KUKA KRL program: MyProgram_035().src

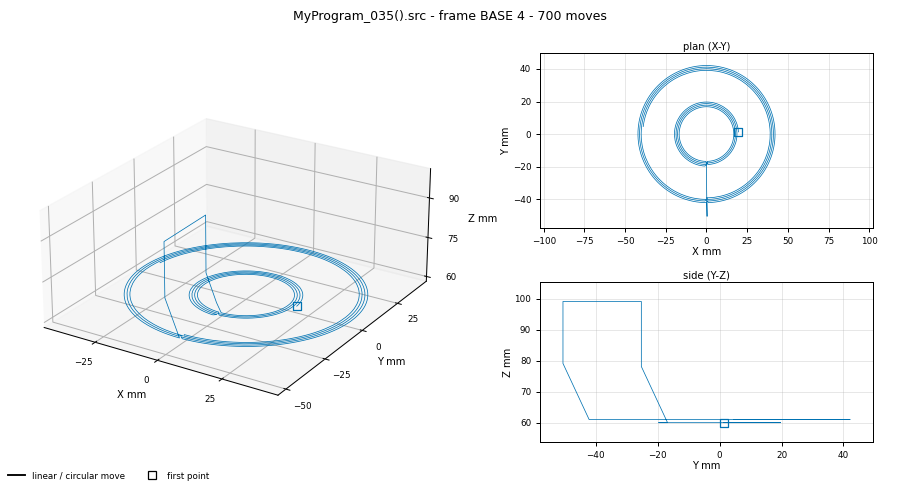
[picture p0: tool path of MyProgram_035().src in frame BASE 4, 700 of 700 moves have a stored position in this frame; points joined in program order, loops and branches not executed]
&ACCESS RVP
&REL 1
&PARAM TEMPLATE = C:\KRC\Roboter\Template\vorgabe
&PARAM EDITMASK = *
DEF MyProgram_035()
; ---- Setting reference (Base) ----
$BASE = BASE_DATA[4]

; --------------------------
; ---- Setting tool (TCP) ----
$TOOL = TOOL_DATA[3]
; --------------------------

$VEL.CP = VEL_APROX_PRINT
Startdeposition()
$VEL.CP = VEL_PRINT
LIN {X 19.6376,Y 1.3472,Z 60,A -3.0599,B 24.8058,C -3.2131,E1 25.1593,E2 -634.5538} C_DIS
LIN {X 19.5136,Y 2.5822,Z 60,A 0.9815,B 24.804,C -3.2283,E1 25.158,E2 -638.6073} C_DIS
LIN {X 19.2505,Y 4.1066,Z 60,A 5.5347,B 24.8023,C -3.2424,E1 25.1555,E2 -643.1673} C_DIS
LIN {X 18.8579,Y 5.6408,Z 60,A 9.7451,B 24.8011,C -3.2522,E1 25.1524,E2 -647.3767} C_DIS
LIN {X 18.3804,Y 7.044,Z 60,A 15.1354,B 24.7983,C -3.2746,E1 25.1472,E2 -652.7902} C_DIS
LIN {X 17.2808,Y 9.4251,Z 60,A 22.0117,B 24.7966,C -3.2881,E1 25.1387,E2 -659.6618} C_DIS
LIN {X 16.4135,Y 10.8654,Z 60,A 26.3437,B 24.7957,C -3.2954,E1 25.1323,E2 -663.9891} C_DIS
LIN {X 15.7405,Y 11.8191,Z 60,A 29.8972,B 24.7945,C -3.305,E1 25.1265,E2 -667.5481} C_DIS
LIN {X 14.7973,Y 12.9806,Z 60,A 34.6576,B 24.7928,C -3.3183,E1 25.1179,E2 -672.3185} C_DIS
LIN {X 13.3773,Y 14.4397,Z 60,A 40.2444,B 24.7917,C -3.3275,E1 25.1068,E2 -677.9036} C_DIS
LIN {X 12.4967,Y 15.2079,Z 60,A 44.9046,B 24.7896,C -3.3443,E1 25.0967,E2 -682.5859} C_DIS
LIN {X 10.1616,Y 16.8582,Z 60,A 52.5619,B 24.7886,C -3.3517,E1 25.0788,E2 -690.2355} C_DIS
LIN {X 8.1073,Y 17.9362,Z 60,A 58.7713,B 24.7881,C -3.3556,E1 25.0633,E2 -696.4376} C_DIS
LIN {X 6.6276,Y 18.5344,Z 60,A 63.8081,B 24.7872,C -3.3628,E1 25.0502,E2 -701.4806} C_DIS
LIN {X 4.5052,Y 19.1613,Z 60,A 69.8964,B 24.787,C -3.3643,E1 25.0338,E2 -707.5628} C_DIS
LIN {X 3.2717,Y 19.4101,Z 60,A 73.6602,B 24.7868,C -3.3663,E1 25.0234,E2 -711.3272} C_DIS
LIN {X 1.6592,Y 19.6136,Z 60,A 78.087,B 24.7869,C -3.365,E1 25.0112,E2 -715.7478} C_DIS
LIN {X 0.0594,Y 19.6839,Z 60,A 83.0982,B 24.7867,C -3.3666,E1 24.9972,E2 -720.7621} C_DIS
LIN {X -1.6521,Y 19.6141,Z 60,A 87.634,B 24.7873,C -3.362,E1 24.9846,E2 -725.2883} C_DIS
LIN {X -2.7882,Y 19.4854,Z 60,A 91.6136,B 24.7871,C -3.3639,E1 24.9735,E2 -729.2752} C_DIS
LIN {X -4.6137,Y 19.1352,Z 60,A 96.3255,B 24.7882,C -3.3554,E1 24.9607,E2 -733.9727} C_DIS
LIN {X -5.6169,Y 18.8652,Z 60,A 99.3541,B 24.7886,C -3.3523,E1 24.9526,E2 -736.9987} C_DIS
LIN {X -6.5937,Y 18.5466,Z 60,A 102.691,B 24.7888,C -3.3506,E1 24.9437,E2 -740.3378} C_DIS
LIN {X -7.8497,Y 18.0506,Z 60,A 106.9874,B 24.7892,C -3.347,E1 24.9327,E2 -744.6356} C_DIS
LIN {X -9.2709,Y 17.3642,Z 60,A 111.6347,B 24.7901,C -3.3399,E1 24.9212,E2 -749.2786} C_DIS
LIN {X -11.1212,Y 16.2413,Z 60,A 118.0633,B 24.7915,C -3.3289,E1 24.9061,E2 -755.7015} C_DIS
LIN {X -12.8725,Y 14.8916,Z 60,A 124.2464,B 24.7934,C -3.3142,E1 24.8927,E2 -761.8727} C_DIS
LIN {X -14.1296,Y 13.7045,Z 60,A 129.3126,B 24.7948,C -3.3026,E1 24.8827,E2 -766.9325} C_DIS
LIN {X -15.2762,Y 12.4134,Z 60,A 134.329,B 24.7964,C -3.2901,E1 24.8736,E2 -771.9417} C_DIS
LIN {X -16.2565,Y 11.099,Z 60,A 139.6568,B 24.7977,C -3.2795,E1 24.865,E2 -777.2704} C_DIS
LIN {X -17.4357,Y 9.1344,Z 60,A 145.3666,B 24.8004,C -3.2573,E1 24.8572,E2 -782.9568} C_DIS
LIN {X -17.9124,Y 8.1607,Z 60,A 149.1514,B 24.8013,C -3.2504,E1 24.8527,E2 -786.7456} C_DIS
LIN {X -18.4403,Y 6.8842,Z 60,A 152.9543,B 24.8028,C -3.2377,E1 24.8489,E2 -790.5395} C_DIS
LIN {X -18.9649,Y 5.2698,Z 60,A 158.2599,B 24.8045,C -3.224,E1 24.8446,E2 -795.8427} C_DIS
LIN {X -19.4015,Y 3.3237,Z 60,A 162.9983,B 24.8071,C -3.2024,E1 24.8419,E2 -800.5574} C_DIS
LIN {X -19.5797,Y 2.0215,Z 60,A 167.8103,B 24.8082,C -3.1938,E1 24.8403,E2 -805.3776} C_DIS
LIN {X -19.6813,Y 0.325,Z 60,A 172.3497,B 24.8102,C -3.177,E1 24.8398,E2 -809.904} C_DIS
LIN {X -19.638,Y -1.3384,Z 60,A 178.2471,B 24.8115,C -3.1657,E1 24.8406,E2 -815.8097} C_DIS
LIN {X -19.2559,Y -4.0801,Z 60,A -173.6054,B 24.8144,C -3.1416,E1 24.8445,E2 -823.9478} C_DIS
LIN {X -18.7721,Y -5.9197,Z 60,A -168.9163,B 24.8167,C -3.1223,E1 24.8481,E2 -828.6178} C_DIS
LIN {X -18.3574,Y -7.1031,Z 60,A -165.3994,B 24.818,C -3.1114,E1 24.8515,E2 -832.1285} C_DIS
LIN {X -17.8438,Y -8.3091,Z 60,A -161.3071,B 24.8191,C -3.102,E1 24.8561,E2 -836.2206} C_DIS
LIN {X -17.2608,Y -9.4618,Z 60,A -157.8679,B 24.8204,C -3.0907,E1 24.8606,E2 -839.6513} C_DIS
LIN {X -16.491,Y -10.7477,Z 60,A -152.7383,B 24.8213,C -3.0828,E1 24.8682,E2 -844.788} C_DIS
LIN {X -15.6196,Y -11.978,Z 60,A -148.4735,B 24.8226,C -3.0719,E1 24.8753,E2 -849.0473} C_DIS
LIN {X -14.4508,Y -13.3656,Z 60,A -143.6937,B 24.8242,C -3.0581,E1 24.8841,E2 -853.8156} C_DIS
LIN {X -13.2063,Y -14.5954,Z 60,A -138.0741,B 24.8251,C -3.0504,E1 24.8955,E2 -859.44} C_DIS
LIN {X -11.8732,Y -15.6997,Z 60,A -133.0339,B 24.8261,C -3.0416,E1 24.9065,E2 -864.4776} C_DIS
LIN {X -10.7284,Y -16.5033,Z 60,A -129.3592,B 24.8271,C -3.0333,E1 24.915,E2 -868.1447} C_DIS
LIN {X -9.4145,Y -17.2865,Z 60,A -124.345,B 24.8274,C -3.0302,E1 24.9272,E2 -873.1664} C_DIS
LIN {X -7.5215,Y -18.1901,Z 60,A -119.2037,B 24.8288,C -3.0183,E1 24.9402,E2 -878.2918} C_DIS
LIN {X -6.3703,Y -18.6242,Z 60,A -114.7625,B 24.8286,C -3.0202,E1 24.9519,E2 -882.7465} C_DIS
LIN {X -4.7968,Y -19.0901,Z 60,A -109.6924,B 24.8286,C -3.0191,E1 24.9656,E2 -887.8218} C_DIS
LIN {X -2.3633,Y -19.5413,Z 60,A -103.3398,B 24.8295,C -3.0117,E1 24.983,E2 -894.1625} C_DIS
LIN {X -0.9908,Y -19.6586,Z 60,A -98.6362,B 24.829,C -3.0163,E1 24.9962,E2 -898.879} C_DIS
LIN {X -0.9908,Y -19.6586,Z 60,A -98.6362,B 24.829,C -3.0163,E1 24.9962,E2 -898.879} C_DIS
Enddeposition()
LIN {X 0.0023,Y -18.7203,Z 60,A -97.1672,B 24.8281,C -3.024,E1 25.0003,E2 -900.3662} C_DIS
Startdeposition()
$VEL.CP = VEL_PRINT
LIN {X -1.3074,Y -18.6798,Z 60,A -102.4252,B 24.829,C -3.0158,E1 24.9856,E2 -895.0876} C_DIS
LIN {X -2.9728,Y -18.4887,Z 60,A -107.3213,B 24.8288,C -3.0182,E1 24.9721,E2 -890.1933} C_DIS
LIN {X -4.4742,Y -18.1833,Z 60,A -112.0588,B 24.8286,C -3.02,E1 24.9591,E2 -885.4543} C_DIS
LIN {X -5.7912,Y -17.8071,Z 60,A -116.0247,B 24.8281,C -3.0241,E1 24.9486,E2 -881.4913} C_DIS
LIN {X -7.2175,Y -17.2787,Z 60,A -120.3356,B 24.8274,C -3.0301,E1 24.9373,E2 -877.1856} C_DIS
LIN {X -8.0909,Y -16.8875,Z 60,A -124.1301,B 24.8275,C -3.0291,E1 24.9277,E2 -873.3792} C_DIS
LIN {X -9.7048,Y -16.0147,Z 60,A -129.7588,B 24.8267,C -3.0366,E1 24.9141,E2 -867.7519} C_DIS
LIN {X -11.1863,Y -15.0175,Z 60,A -135.1337,B 24.8256,C -3.0458,E1 24.9018,E2 -862.3804} C_DIS
LIN {X -12.5346,Y -13.912,Z 60,A -140.552,B 24.8245,C -3.0554,E1 24.8903,E2 -856.9639} C_DIS
LIN {X -13.7315,Y -12.7322,Z 60,A -145.7596,B 24.8233,C -3.0658,E1 24.8802,E2 -851.7589} C_DIS
LIN {X -14.7656,Y -11.5172,Z 60,A -151.4599,B 24.8224,C -3.074,E1 24.8703,E2 -846.0516} C_DIS
LIN {X -16.3018,Y -9.215,Z 60,A -159.7556,B 24.8198,C -3.096,E1 24.8581,E2 -837.7662} C_DIS
LIN {X -17.2394,Y -7.3112,Z 60,A -165.587,B 24.8175,C -3.1159,E1 24.8513,E2 -831.9507} C_DIS
LIN {X -17.7997,Y -5.8135,Z 60,A -170.3075,B 24.8157,C -3.1305,E1 24.8469,E2 -827.2382} C_DIS
LIN {X -18.199,Y -4.4089,Z 60,A -175.0055,B 24.8143,C -3.143,E1 24.8436,E2 -822.5429} C_DIS
LIN {X -18.4596,Y -3.1467,Z 60,A -178.7025,B 24.8128,C -3.1556,E1 24.8417,E2 -818.8542} C_DIS
LIN {X -18.6406,Y -1.7791,Z 60,A 176.7274,B 24.8113,C -3.1675,E1 24.8402,E2 -814.2853} C_DIS
LIN {X -18.7241,Y 0.0458,Z 60,A 171.3284,B 24.8092,C -3.1854,E1 24.8398,E2 -808.8967} C_DIS
LIN {X -18.6556,Y 1.6172,Z 60,A 166.2101,B 24.8075,C -3.1995,E1 24.8407,E2 -803.7814} C_DIS
LIN {X -18.4421,Y 3.248,Z 60,A 161.0802,B 24.8056,C -3.2149,E1 24.8429,E2 -798.6578} C_DIS
LIN {X -18.0417,Y 5.0134,Z 60,A 155.5596,B 24.8035,C -3.2319,E1 24.8466,E2 -793.1458} C_DIS
LIN {X -17.4548,Y 6.7805,Z 60,A 150.3263,B 24.8013,C -3.2504,E1 24.8514,E2 -787.927} C_DIS
LIN {X -17.0487,Y 7.7456,Z 60,A 146.7149,B 24.8003,C -3.2585,E1 24.8555,E2 -784.3152} C_DIS
LIN {X -16.289,Y 9.2368,Z 60,A 140.7953,B 24.7988,C -3.2705,E1 24.8634,E2 -778.3931} C_DIS
LIN {X -15.1642,Y 10.9866,Z 60,A 135.0172,B 24.7964,C -3.2895,E1 24.8724,E2 -772.6318} C_DIS
LIN {X -14.128,Y 12.2906,Z 60,A 129.8754,B 24.7949,C -3.3021,E1 24.8816,E2 -767.4966} C_DIS
LIN {X -12.9816,Y 13.4956,Z 60,A 124.7751,B 24.7934,C -3.314,E1 24.8916,E2 -762.403} C_DIS
LIN {X -11.9092,Y 14.451,Z 60,A 120.0573,B 24.7923,C -3.3223,E1 24.9017,E2 -757.6868} C_DIS
LIN {X -10.4305,Y 15.552,Z 60,A 114.9908,B 24.7907,C -3.3356,E1 24.9131,E2 -752.6347} C_DIS
LIN {X -9.0786,Y 16.3779,Z 60,A 109.8141,B 24.7898,C -3.3426,E1 24.9256,E2 -747.4592} C_DIS
LIN {X -7.5346,Y 17.1427,Z 60,A 104.2599,B 24.7889,C -3.3492,E1 24.9397,E2 -741.907} C_DIS
LIN {X -5.6024,Y 17.8678,Z 60,A 97.8473,B 24.788,C -3.3563,E1 24.9566,E2 -735.499} C_DIS
LIN {X -3.4857,Y 18.3984,Z 60,A 91.502,B 24.7871,C -3.3638,E1 24.9738,E2 -729.1635} C_DIS
LIN {X -1.8213,Y 18.6369,Z 60,A 86.2377,B 24.7868,C -3.3661,E1 24.9884,E2 -723.901} C_DIS
LIN {X -0.1445,Y 18.7253,Z 60,A 81.1999,B 24.7865,C -3.3681,E1 25.0025,E2 -718.8673} C_DIS
LIN {X 1.3917,Y 18.6736,Z 60,A 76.1915,B 24.7868,C -3.3664,E1 25.0164,E2 -713.8567} C_DIS
LIN {X 3.3103,Y 18.4309,Z 60,A 70.337,B 24.7869,C -3.3651,E1 25.0326,E2 -708.0047} C_DIS
LIN {X 5.2188,Y 17.9836,Z 60,A 64.4223,B 24.7873,C -3.3621,E1 25.0485,E2 -702.0919} C_DIS
LIN {X 6.6991,Y 17.4858,Z 60,A 60.4332,B 24.7871,C -3.3634,E1 25.059,E2 -698.1141} C_DIS
LIN {X 7.7404,Y 17.051,Z 60,A 56.5752,B 24.788,C -3.3568,E1 25.0689,E2 -694.2498} C_DIS
LIN {X 8.9291,Y 16.4598,Z 60,A 52.631,B 24.7885,C -3.3526,E1 25.0787,E2 -690.3065} C_DIS
LIN {X 10.4844,Y 15.515,Z 60,A 45.6574,B 24.7909,C -3.3336,E1 25.0951,E2 -683.3106} C_DIS
LIN {X 12.3955,Y 14.0359,Z 60,A 39.895,B 24.791,C -3.3329,E1 25.1075,E2 -677.5682} C_DIS
LIN {X 13.3706,Y 13.1097,Z 60,A 35.602,B 24.7922,C -3.3231,E1 25.116,E2 -673.27} C_DIS
LIN {X 14.248,Y 12.1511,Z 60,A 31.5215,B 24.7934,C -3.3135,E1 25.1236,E2 -669.185} C_DIS
LIN {X 15.218,Y 10.912,Z 60,A 26.5171,B 24.7951,C -3.3005,E1 25.132,E2 -664.1737} C_DIS
LIN {X 16.1415,Y 9.4927,Z 60,A 21.3329,B 24.7967,C -3.2873,E1 25.1396,E2 -658.9845} C_DIS
LIN {X 16.9883,Y 7.8764,Z 60,A 15.6192,B 24.7987,C -3.2711,E1 25.1467,E2 -653.2629} C_DIS
LIN {X 17.5234,Y 6.6008,Z 60,A 11.2667,B 24.8003,C -3.2581,E1 25.1511,E2 -648.9037} C_DIS
LIN {X 18.1197,Y 4.7245,Z 60,A 5.6681,B 24.802,C -3.2442,E1 25.1555,E2 -643.3042} C_DIS
LIN {X 18.4918,Y 2.9509,Z 60,A -0.4867,B 24.8048,C -3.222,E1 25.1585,E2 -637.1327} C_DIS
LIN {X 18.704,Y 0.8956,Z 60,A -6.4334,B 24.8067,C -3.2058,E1 25.1597,E2 -631.1831} C_DIS
LIN {X 18.7034,Y -0.9078,Z 60,A -11.3548,B 24.8081,C -3.1941,E1 25.1594,E2 -626.2631} C_DIS
LIN {X 18.5918,Y -2.2333,Z 60,A -15.3986,B 24.8096,C -3.1816,E1 25.1583,E2 -622.2138} C_DIS
LIN {X 18.3067,Y -3.9382,Z 60,A -20.8999,B 24.8118,C -3.1633,E1 25.1555,E2 -616.7012} C_DIS
LIN {X 17.8954,Y -5.5135,Z 60,A -25.9073,B 24.8137,C -3.1478,E1 25.1516,E2 -611.6858} C_DIS
LIN {X 17.4696,Y -6.7422,Z 60,A -29.5087,B 24.8147,C -3.1393,E1 25.1481,E2 -608.0844} C_DIS
LIN {X 17.0745,Y -7.6882,Z 60,A -32.8176,B 24.816,C -3.1286,E1 25.1444,E2 -604.768} C_DIS
LIN {X 16.3664,Y -9.0987,Z 60,A -37.4347,B 24.8174,C -3.1166,E1 25.1384,E2 -600.147} C_DIS
LIN {X 15.6588,Y -10.2663,Z 60,A -40.6077,B 24.8177,C -3.114,E1 25.1338,E2 -596.9839} C_DIS
LIN {X 15.164,Y -10.9869,Z 60,A -44.1903,B 24.8195,C -3.0988,E1 25.128,E2 -593.3828} C_DIS
LIN {X 14.3596,Y -12.0187,Z 60,A -48.9247,B 24.8214,C -3.0823,E1 25.1196,E2 -588.6312} C_DIS
LIN {X 13.0169,Y -13.4616,Z 60,A -54.4704,B 24.8226,C -3.072,E1 25.1088,E2 -583.0849} C_DIS
LIN {X 11.6539,Y -14.6571,Z 60,A -59.971,B 24.8239,C -3.0604,E1 25.097,E2 -577.5777} C_DIS
LIN {X 10.4375,Y -15.5473,Z 60,A -64.481,B 24.8249,C -3.0521,E1 25.0867,E2 -573.0636} C_DIS
LIN {X 9.1733,Y -16.3247,Z 60,A -69.5837,B 24.8263,C -3.0397,E1 25.0744,E2 -567.947} C_DIS
LIN {X 7.4057,Y -17.1987,Z 60,A -75.1897,B 24.827,C -3.0338,E1 25.0602,E2 -562.3413} C_DIS
LIN {X 5.9027,Y -17.7706,Z 60,A -79.0907,B 24.8269,C -3.035,E1 25.05,E2 -558.4513} C_DIS
LIN {X 4.7432,Y -18.1147,Z 60,A -84.1337,B 24.8284,C -3.0215,E1 25.0364,E2 -553.3845} C_DIS
LIN {X 2.5879,Y -18.546,Z 60,A -90.5837,B 24.8288,C -3.0183,E1 25.0186,E2 -546.9337} C_DIS
LIN {X 0.9263,Y -18.7024,Z 60,A -95.0252,B 24.8285,C -3.0203,E1 25.0063,E2 -542.4991} C_DIS
LIN {X 0.9263,Y -18.7024,Z 60,A -95.0252,B 24.8285,C -3.0203,E1 25.0063,E2 -542.4991} C_DIS
Enddeposition()
LIN {X 0.0155,Y -17.7649,Z 60,A -97.9923,B 24.8268,C -3.0353,E1 24.9981,E2 -539.5681} C_DIS
Startdeposition()
$VEL.CP = VEL_PRINT
LIN {X 0.9859,Y -17.7401,Z 60,A -92.6978,B 24.8252,C -3.0497,E1 25.013,E2 -544.8957} C_DIS
LIN {X 2.8059,Y -17.5446,Z 60,A -86.903,B 24.8248,C -3.0527,E1 25.029,E2 -550.6929} C_DIS
LIN {X 4.419,Y -17.2087,Z 60,A -82.0027,B 24.8246,C -3.0547,E1 25.0423,E2 -555.5912} C_DIS
LIN {X 5.782,Y -16.8003,Z 60,A -76.9277,B 24.8236,C -3.0635,E1 25.0559,E2 -560.6777} C_DIS
LIN {X 7.3313,Y -16.1845,Z 60,A -71.5706,B 24.8227,C -3.0711,E1 25.0696,E2 -566.0401} C_DIS
LIN {X 8.8093,Y -15.4301,Z 60,A -66.2939,B 24.8217,C -3.0795,E1 25.0826,E2 -571.3216} C_DIS
LIN {X 10.1378,Y -14.5916,Z 60,A -61.2643,B 24.8206,C -3.0889,E1 25.0943,E2 -576.3567} C_DIS
LIN {X 11.4347,Y -13.5993,Z 60,A -55.9441,B 24.8193,C -3.1005,E1 25.1059,E2 -581.6845} C_DIS
LIN {X 12.6468,Y -12.4798,Z 60,A -50.6998,B 24.8179,C -3.1122,E1 25.1164,E2 -586.9349} C_DIS
LIN {X 13.7519,Y -11.2508,Z 60,A -45.3857,B 24.8163,C -3.1254,E1 25.1261,E2 -592.2562} C_DIS
LIN {X 14.48,Y -10.2967,Z 60,A -41.3387,B 24.8149,C -3.1372,E1 25.1328,E2 -596.3116} C_DIS
LIN {X 15.3947,Y -8.871,Z 60,A -36.4867,B 24.8138,C -3.147,E1 25.1398,E2 -601.1622} C_DIS
LIN {X 15.9584,Y -7.8103,Z 60,A -32.2515,B 24.8121,C -3.1614,E1 25.1452,E2 -605.4089} C_DIS
LIN {X 16.6204,Y -6.2801,Z 60,A -26.9211,B 24.8102,C -3.1769,E1 25.1508,E2 -610.7467} C_DIS
LIN {X 17.1291,Y -4.7193,Z 60,A -21.6748,B 24.8083,C -3.1926,E1 25.155,E2 -616.0002} C_DIS
LIN {X 17.4958,Y -3.0967,Z 60,A -16.5828,B 24.8066,C -3.2067,E1 25.1578,E2 -621.096} C_DIS
LIN {X 17.6916,Y -1.6394,Z 60,A -11.8559,B 24.8048,C -3.2214,E1 25.1593,E2 -625.8297} C_DIS
LIN {X 17.7588,Y -0.5555,Z 60,A -7.9269,B 24.803,C -3.2362,E1 25.1598,E2 -629.7704} C_DIS
LIN {X 17.7238,Y 1.2423,Z 60,A -2.3861,B 24.8011,C -3.2518,E1 25.1591,E2 -635.3153} C_DIS
LIN {X 17.5367,Y 2.8563,Z 60,A 2.8447,B 24.7991,C -3.2677,E1 25.1571,E2 -640.553} C_DIS
LIN {X 17.0145,Y 5.1185,Z 60,A 11.2683,B 24.7954,C -3.2982,E1 25.151,E2 -649.0004} C_DIS
LIN {X 16.2621,Y 7.1575,Z 60,A 17.5108,B 24.7937,C -3.3111,E1 25.1444,E2 -655.239} C_DIS
LIN {X 15.4456,Y 8.7823,Z 60,A 23.048,B 24.7922,C -3.3238,E1 25.1371,E2 -660.7772} C_DIS
LIN {X 14.5893,Y 10.1411,Z 60,A 28.1705,B 24.7906,C -3.3361,E1 25.1292,E2 -665.9036} C_DIS
LIN {X 13.5375,Y 11.5077,Z 60,A 33.9985,B 24.7887,C -3.3511,E1 25.1189,E2 -671.7401} C_DIS
LIN {X 12.2964,Y 12.8253,Z 60,A 39.5523,B 24.7875,C -3.3609,E1 25.108,E2 -677.2934} C_DIS
LIN {X 11.0852,Y 13.8857,Z 60,A 44.6875,B 24.7863,C -3.37,E1 25.097,E2 -682.4306} C_DIS
LIN {X 9.7729,Y 14.8385,Z 60,A 49.6403,B 24.7855,C -3.3764,E1 25.0857,E2 -687.3815} C_DIS
LIN {X 8.5658,Y 15.5668,Z 60,A 54.8686,B 24.7841,C -3.3875,E1 25.073,E2 -692.6209} C_DIS
LIN {X 6.8255,Y 16.4041,Z 60,A 60.4967,B 24.7837,C -3.3902,E1 25.0587,E2 -698.2412} C_DIS
LIN {X 5.1776,Y 16.9963,Z 60,A 66.6407,B 24.7827,C -3.398,E1 25.0424,E2 -704.392} C_DIS
LIN {X 3.6988,Y 17.3781,Z 60,A 70.4944,B 24.7833,C -3.3937,E1 25.032,E2 -708.2302} C_DIS
LIN {X 2.1269,Y 17.6396,Z 60,A 76.3306,B 24.7825,C -3.3994,E1 25.0158,E2 -714.0744} C_DIS
LIN {X 0.5104,Y 17.7602,Z 60,A 81.5201,B 24.7825,C -3.399,E1 25.0014,E2 -719.2612} C_DIS
LIN {X -1.0448,Y 17.7365,Z 60,A 86.6495,B 24.7827,C -3.3981,E1 24.9871,E2 -724.3894} C_DIS
LIN {X -2.7119,Y 17.5595,Z 60,A 92.0361,B 24.7831,C -3.3948,E1 24.9722,E2 -729.772} C_DIS
LIN {X -4.288,Y 17.2422,Z 60,A 97.2456,B 24.7837,C -3.3904,E1 24.958,E2 -734.9777} C_DIS
LIN {X -5.3974,Y 16.9275,Z 60,A 101.2596,B 24.784,C -3.3877,E1 24.9473,E2 -738.9922} C_DIS
LIN {X -7.2707,Y 16.2117,Z 60,A 107.9497,B 24.785,C -3.3798,E1 24.9301,E2 -745.6788} C_DIS
LIN {X -8.9768,Y 15.3334,Z 60,A 112.926,B 24.787,C -3.3645,E1 24.9179,E2 -750.6325} C_DIS
LIN {X -9.8381,Y 14.7955,Z 60,A 116.3784,B 24.7877,C -3.3592,E1 24.9098,E2 -754.0832} C_DIS
LIN {X -10.8797,Y 14.0472,Z 60,A 121.1427,B 24.7884,C -3.3532,E1 24.8991,E2 -758.8504} C_DIS
LIN {X -12.1249,Y 12.9875,Z 60,A 126.3848,B 24.7899,C -3.3415,E1 24.8882,E2 -764.0852} C_DIS
LIN {X -13.2496,Y 11.838,Z 60,A 131.6257,B 24.7915,C -3.3292,E1 24.8782,E2 -769.3195} C_DIS
LIN {X -14.2665,Y 10.5908,Z 60,A 136.8701,B 24.7931,C -3.316,E1 24.8693,E2 -774.5573} C_DIS
LIN {X -15.1697,Y 9.2502,Z 60,A 141.9423,B 24.795,C -3.3014,E1 24.8616,E2 -779.6201} C_DIS
LIN {X -15.8004,Y 8.1265,Z 60,A 145.8324,B 24.7965,C -3.2888,E1 24.8565,E2 -783.5006} C_DIS
LIN {X -16.3391,Y 6.9794,Z 60,A 150.1115,B 24.7979,C -3.2775,E1 24.8516,E2 -787.776} C_DIS
LIN {X -16.8888,Y 5.518,Z 60,A 155.9725,B 24.7995,C -3.2648,E1 24.8462,E2 -793.6399} C_DIS
LIN {X -17.3922,Y 3.6333,Z 60,A 161.8048,B 24.802,C -3.2441,E1 24.8425,E2 -799.4568} C_DIS
LIN {X -17.6508,Y 2.0329,Z 60,A 167.1192,B 24.804,C -3.2281,E1 24.8404,E2 -804.7647} C_DIS
LIN {X -17.764,Y 0.3659,Z 60,A 172.7123,B 24.806,C -3.2119,E1 24.8398,E2 -810.3525} C_DIS
LIN {X -17.7434,Y -0.9139,Z 60,A 176.7278,B 24.8076,C -3.1989,E1 24.8402,E2 -814.3608} C_DIS
LIN {X -17.5864,Y -2.5306,Z 60,A -177.5893,B 24.8093,C -3.1841,E1 24.8422,E2 -820.0423} C_DIS
LIN {X -17.0785,Y -4.8999,Z 60,A -170.2362,B 24.8123,C -3.1595,E1 24.847,E2 -827.3795} C_DIS
LIN {X -16.569,Y -6.4147,Z 60,A -165.0333,B 24.814,C -3.145,E1 24.852,E2 -832.577} C_DIS
LIN {X -16.046,Y -7.6299,Z 60,A -161.0987,B 24.8155,C -3.1322,E1 24.8565,E2 -836.5026} C_DIS
LIN {X -15.4602,Y -8.7566,Z 60,A -156.7355,B 24.8167,C -3.1223,E1 24.8623,E2 -840.8652} C_DIS
LIN {X -14.767,Y -9.88,Z 60,A -151.9945,B 24.8178,C -3.1134,E1 24.8695,E2 -845.6087} C_DIS
LIN {X -13.685,Y -11.3319,Z 60,A -146.3624,B 24.8194,C -3.0992,E1 24.8792,E2 -851.2332} C_DIS
LIN {X -12.5761,Y -12.5515,Z 60,A -141.0401,B 24.8207,C -3.088,E1 24.8895,E2 -856.552} C_DIS
LIN {X -11.35,Y -13.67,Z 60,A -135.6464,B 24.8219,C -3.0782,E1 24.9008,E2 -861.9433} C_DIS
LIN {X -10.2593,Y -14.5066,Z 60,A -131.2588,B 24.8227,C -3.0706,E1 24.9107,E2 -866.3283} C_DIS
LIN {X -8.9005,Y -15.3776,Z 60,A -125.9838,B 24.8236,C -3.0635,E1 24.9233,E2 -871.6026} C_DIS
LIN {X -7.3207,Y -16.1892,Z 60,A -120.3803,B 24.8244,C -3.0563,E1 24.9374,E2 -877.2034} C_DIS
LIN {X -6.0534,Y -16.7038,Z 60,A -116.2283,B 24.825,C -3.051,E1 24.9482,E2 -881.3515} C_DIS
LIN {X -4.626,Y -17.1546,Z 60,A -111.0042,B 24.8251,C -3.0499,E1 24.9622,E2 -886.5816} C_DIS
LIN {X -3.0319,Y -17.5074,Z 60,A -105.7637,B 24.8254,C -3.0477,E1 24.9765,E2 -891.8228} C_DIS
LIN {X -1.4921,Y -17.7046,Z 60,A -100.694,B 24.8254,C -3.0477,E1 24.9906,E2 -896.8952} C_DIS
LIN {X 0.0155,Y -17.7649,Z 60,A -97.9922,B 24.8268,C -3.0353,E1 24.9981,E2 -899.5681} C_DIS
Enddeposition()
LIN {X 0.0155,Y -17.7649,Z 60,A -97.9922,B 24.8268,C -3.0353,E1 24.9981,E2 -899.5681} C_DIS
Startdeposition()
$VEL.CP = VEL_PRINT
LIN {X -0.4182,Y -16.8044,Z 60,A -100.0886,B 24.8253,C -3.0484,E1 24.9923,E2 -897.5028} C_DIS
LIN {X -1.9453,Y -16.6964,Z 60,A -105.0785,B 24.8251,C -3.05,E1 24.9785,E2 -892.514} C_DIS
LIN {X -3.3845,Y -16.4651,Z 60,A -110.07,B 24.825,C -3.0515,E1 24.9647,E2 -887.521} C_DIS
LIN {X -4.8682,Y -16.089,Z 60,A -115.4755,B 24.8247,C -3.0539,E1 24.9502,E2 -882.1125} C_DIS
LIN {X -6.509,Y -15.497,Z 60,A -119.9286,B 24.8233,C -3.0659,E1 24.9386,E2 -877.6791} C_DIS
LIN {X -7.8899,Y -14.8426,Z 60,A -125.1752,B 24.8226,C -3.0716,E1 24.9254,E2 -872.4327} C_DIS
LIN {X -9.2418,Y -14.0409,Z 60,A -130.6854,B 24.8218,C -3.0784,E1 24.9121,E2 -866.9222} C_DIS
LIN {X -10.5128,Y -13.1165,Z 60,A -136.1827,B 24.8209,C -3.0867,E1 24.8997,E2 -861.4255} C_DIS
LIN {X -11.2936,Y -12.4505,Z 60,A -140.4226,B 24.8204,C -3.0906,E1 24.8908,E2 -857.1782} C_DIS
LIN {X -12.2148,Y -11.548,Z 60,A -145.3533,B 24.8196,C -3.0979,E1 24.8811,E2 -852.2439} C_DIS
LIN {X -13.2504,Y -10.344,Z 60,A -150.6717,B 24.8181,C -3.1105,E1 24.8717,E2 -846.9309} C_DIS
LIN {X -13.8659,Y -9.5027,Z 60,A -153.9519,B 24.817,C -3.1199,E1 24.8664,E2 -843.6571} C_DIS
LIN {X -14.7157,Y -8.1246,Z 60,A -158.512,B 24.815,C -3.1367,E1 24.8599,E2 -839.1139} C_DIS
LIN {X -15.0377,Y -7.5116,Z 60,A -161.937,B 24.8146,C -3.1401,E1 24.8555,E2 -835.6786} C_DIS
LIN {X -15.6146,Y -6.2234,Z 60,A -167.1215,B 24.8131,C -3.1525,E1 24.8498,E2 -830.4951} C_DIS
LIN {X -16.144,Y -4.6824,Z 60,A -172.7406,B 24.8112,C -3.1684,E1 24.8451,E2 -824.882} C_DIS
LIN {X -16.5214,Y -3.0984,Z 60,A -178.1227,B 24.8092,C -3.1854,E1 24.842,E2 -819.5089} C_DIS
LIN {X -16.7334,Y -1.5956,Z 60,A 176.546,B 24.8073,C -3.2009,E1 24.8402,E2 -814.1829} C_DIS
LIN {X -16.8079,Y -0.1139,Z 60,A 171.6038,B 24.8054,C -3.2169,E1 24.8398,E2 -809.2491} C_DIS
LIN {X -16.7476,Y 1.4383,Z 60,A 166.1857,B 24.8034,C -3.2331,E1 24.8407,E2 -803.8373} C_DIS
LIN {X -16.5501,Y 2.9418,Z 60,A 162.0715,B 24.8011,C -3.2515,E1 24.8423,E2 -799.7428} C_DIS
LIN {X -16.1968,Y 4.4952,Z 60,A 156.6454,B 24.7991,C -3.2682,E1 24.8457,E2 -794.3248} C_DIS
LIN {X -15.9948,Y 5.1686,Z 60,A 153.1141,B 24.7985,C -3.2728,E1 24.8486,E2 -790.7842} C_DIS
LIN {X -15.4869,Y 6.5352,Z 60,A 148.1021,B 24.7967,C -3.2874,E1 24.8538,E2 -785.7792} C_DIS
LIN {X -14.7754,Y 8.0154,Z 60,A 143.6108,B 24.7944,C -3.3062,E1 24.8593,E2 -781.3089} C_DIS
LIN {X -13.9899,Y 9.319,Z 60,A 138.2998,B 24.7926,C -3.3202,E1 24.867,E2 -776.0042} C_DIS
LIN {X -13.4314,Y 10.1073,Z 60,A 133.758,B 24.7919,C -3.3255,E1 24.8745,E2 -771.4528} C_DIS
LIN {X -12.4167,Y 11.3305,Z 60,A 128.4235,B 24.7902,C -3.3391,E1 24.8842,E2 -766.1269} C_DIS
LIN {X -11.168,Y 12.5634,Z 60,A 123.5433,B 24.7881,C -3.3562,E1 24.894,E2 -761.2674} C_DIS
LIN {X -9.9444,Y 13.5524,Z 60,A 118.2043,B 24.7866,C -3.3675,E1 24.9056,E2 -755.9355} C_DIS
LIN {X -8.6339,Y 14.423,Z 60,A 112.715,B 24.7854,C -3.3771,E1 24.9183,E2 -750.4512} C_DIS
LIN {X -7.2839,Y 15.1493,Z 60,A 107.5379,B 24.7843,C -3.3859,E1 24.9311,E2 -745.2805} C_DIS
LIN {X -6.6823,Y 15.4237,Z 60,A 104.0355,B 24.7845,C -3.3842,E1 24.94,E2 -741.7656} C_DIS
LIN {X -5.2567,Y 15.966,Z 60,A 99.1574,B 24.7835,C -3.3919,E1 24.9528,E2 -736.8963} C_DIS
LIN {X -3.7006,Y 16.3971,Z 60,A 94.4476,B 24.7824,C -3.4008,E1 24.9655,E2 -732.2006} C_DIS
LIN {X -2.6638,Y 16.5974,Z 60,A 90.1413,B 24.7824,C -3.4002,E1 24.9773,E2 -727.8884} C_DIS
LIN {X -1.4397,Y 16.7475,Z 60,A 85.454,B 24.7824,C -3.4,E1 24.9904,E2 -723.198} C_DIS
LIN {X 0.1108,Y 16.8092,Z 60,A 80.1673,B 24.7823,C -3.4013,E1 25.0051,E2 -717.9141} C_DIS
LIN {X 1.6407,Y 16.7291,Z 60,A 74.9464,B 24.7823,C -3.4011,E1 25.0196,E2 -712.6953} C_DIS
LIN {X 3.1559,Y 16.5105,Z 60,A 69.8342,B 24.7825,C -3.4,E1 25.0337,E2 -707.5857} C_DIS
LIN {X 4.8288,Y 16.1007,Z 60,A 65.1742,B 24.782,C -3.4038,E1 25.0463,E2 -702.9419} C_DIS
LIN {X 6.1616,Y 15.6393,Z 60,A 60.5752,B 24.7823,C -3.4011,E1 25.0584,E2 -698.3456} C_DIS
LIN {X 6.7427,Y 15.3976,Z 60,A 56.9222,B 24.7838,C -3.3892,E1 25.0678,E2 -694.6728} C_DIS
LIN {X 8.1232,Y 14.7166,Z 60,A 51.8212,B 24.7846,C -3.3835,E1 25.0804,E2 -689.5725} C_DIS
LIN {X 9.4411,Y 13.9077,Z 60,A 46.427,B 24.7857,C -3.3746,E1 25.0931,E2 -684.1749} C_DIS
LIN {X 10.7448,Y 12.9269,Z 60,A 40.9601,B 24.7869,C -3.3655,E1 25.1051,E2 -678.7066} C_DIS
LIN {X 11.8825,Y 11.8902,Z 60,A 35.723,B 24.7882,C -3.355,E1 25.1157,E2 -673.4663} C_DIS
LIN {X 12.9872,Y 10.6721,Z 60,A 31.3156,B 24.7886,C -3.3518,E1 25.1238,E2 -669.0711} C_DIS
LIN {X 13.9226,Y 9.419,Z 60,A 26.1217,B 24.7901,C -3.3402,E1 25.1325,E2 -663.8745} C_DIS
LIN {X 14.311,Y 8.8182,Z 60,A 22.5254,B 24.792,C -3.3249,E1 25.1379,E2 -660.2599} C_DIS
LIN {X 15.0137,Y 7.5602,Z 60,A 17.6155,B 24.7937,C -3.3119,E1 25.1443,E2 -655.345} C_DIS
LIN {X 15.6225,Y 6.204,Z 60,A 12.4644,B 24.7955,C -3.2971,E1 25.1499,E2 -650.1871} C_DIS
LIN {X 16.1502,Y 4.6614,Z 60,A 6.9084,B 24.7975,C -3.2809,E1 25.1546,E2 -644.6244} C_DIS
LIN {X 16.5275,Y 3.0669,Z 60,A 1.5452,B 24.7993,C -3.266,E1 25.1577,E2 -639.2571} C_DIS
LIN {X 16.7287,Y 1.645,Z 60,A -3.5142,B 24.8014,C -3.2497,E1 25.1593,E2 -634.1887} C_DIS
LIN {X 16.8079,Y 0.1139,Z 60,A -2.9189,B 24.7971,C -3.2844,E1 25.1593,E2 -634.8628} C_DIS
LIN {X 16.78,Y -0.9888,Z 60,A -11.1568,B 24.8034,C -3.2332,E1 25.1595,E2 -626.5526} C_DIS
LIN {X 16.6193,Y -2.5212,Z 60,A -16.3228,B 24.8053,C -3.2176,E1 25.158,E2 -621.3801} C_DIS
LIN {X 16.3598,Y -3.8595,Z 60,A -20.2996,B 24.8063,C -3.209,E1 25.1559,E2 -617.4062} C_DIS
LIN {X 16.1435,Y -4.6841,Z 60,A -25.1368,B 24.8094,C -3.1835,E1 25.1524,E2 -612.5365} C_DIS
LIN {X 15.608,Y -6.24,Z 60,A -30.6387,B 24.8113,C -3.1676,E1 25.147,E2 -607.0277} C_DIS
LIN {X 14.9442,Y -7.6964,Z 60,A -36.112,B 24.8132,C -3.1517,E1 25.1403,E2 -601.5459} C_DIS
LIN {X 14.0486,Y -9.2303,Z 60,A -40.8888,B 24.814,C -3.1454,E1 25.1335,E2 -596.7786} C_DIS
LIN {X 13.1309,Y -10.4948,Z 60,A -46.1884,B 24.8156,C -3.1315,E1 25.1248,E2 -591.4716} C_DIS
LIN {X 12.76,Y -10.9426,Z 60,A -49.3308,B 24.8173,C -3.1172,E1 25.119,E2 -588.3097} C_DIS
LIN {X 11.7052,Y -12.0643,Z 60,A -54.5453,B 24.8187,C -3.105,E1 25.1088,E2 -583.0885} C_DIS
LIN {X 10.4015,Y -13.2048,Z 60,A -59.0909,B 24.819,C -3.1025,E1 25.0992,E2 -578.5546} C_DIS
LIN {X 9.15,Y -14.1009,Z 60,A -64.4783,B 24.8204,C -3.091,E1 25.087,E2 -573.1588} C_DIS
LIN {X 7.8217,Y -14.8786,Z 60,A -69.6179,B 24.8214,C -3.0825,E1 25.0746,E2 -568.0146} C_DIS
LIN {X 6.8071,Y -15.3695,Z 60,A -74.7944,B 24.8231,C -3.0673,E1 25.0614,E2 -562.8152} C_DIS
LIN {X 5.3183,Y -15.9455,Z 60,A -79.994,B 24.8237,C -3.062,E1 25.0478,E2 -557.6138} C_DIS
LIN {X 3.7032,Y -16.3965,Z 60,A -84.711,B 24.8237,C -3.0626,E1 25.0351,E2 -552.9058} C_DIS
LIN {X 2.0927,Y -16.6785,Z 60,A -90.2218,B 24.8241,C -3.0588,E1 25.0199,E2 -547.3918} C_DIS
LIN {X 0.5208,Y -16.8013,Z 60,A -95.4727,B 24.8243,C -3.0571,E1 25.0053,E2 -542.1392} C_DIS
LIN {X 0.5208,Y -16.8013,Z 60,A -95.4727,B 24.8243,C -3.0571,E1 25.0053,E2 -542.1392} C_DIS
Enddeposition()
LIN {X 0.0049,Y -18.9215,Z 64.5315,A -97.7532,B 24.8255,C -3.0471,E1 24.9988,E2 -539.8353} C_DIS
LIN {X -0.0535,Y -25.2605,Z 78.1262,A -97.7145,B 24.8273,C -3.0309,E1 24.9988,E2 -539.8353} C_DIS
LIN {X -0.0535,Y -25.2605,Z 99.1262,A -98.0626,B 24.8102,C -3.177,E1 24.9988,E2 -539.8353} C_DIS
LIN {X 0.3545,Y -50.566,Z 99.1262,A -95.6021,B 24.8565,C -2.7639,E1 25.003,E2 -541.3121} C_DIS
LIN {X 0.3545,Y -50.566,Z 79.1262,A -95.2709,B 24.8707,C -2.6246,E1 25.003,E2 -541.3121} C_DIS
LIN {X 0.2495,Y -44.2276,Z 65.5315,A -95.3053,B 24.8692,C -2.6391,E1 25.003,E2 -541.3121} C_DIS
LIN {X 0.2145,Y -42.1147,Z 61,A -95.3182,B 24.8687,C -2.6445,E1 25.003,E2 -541.3121} C_DIS
Startdeposition()
$VEL.CP = VEL_PRINT
LIN {X -2.0197,Y -42.0691,Z 61,A -99.6024,B 24.8705,C -2.6259,E1 24.9909,E2 -536.9833} C_DIS
LIN {X -4.1283,Y -41.915,Z 61,A -102.5495,B 24.8706,C -2.625,E1 24.9827,E2 -534.0327} C_DIS
LIN {X -6.1335,Y -41.6686,Z 61,A -105.3167,B 24.8706,C -2.6253,E1 24.975,E2 -531.264} C_DIS
LIN {X -8.1707,Y -41.3175,Z 61,A -108.1315,B 24.8705,C -2.6262,E1 24.9673,E2 -528.4485} C_DIS
LIN {X -10.2338,Y -40.8556,Z 61,A -110.9773,B 24.8703,C -2.6281,E1 24.9595,E2 -525.6032} C_DIS
LIN {X -12.2262,Y -40.3043,Z 61,A -113.7943,B 24.8701,C -2.6298,E1 24.952,E2 -522.7859} C_DIS
LIN {X -14.2332,Y -39.6397,Z 61,A -116.8748,B 24.8701,C -2.6294,E1 24.9438,E2 -519.6985} C_DIS
LIN {X -16.5508,Y -38.7293,Z 61,A -120.1052,B 24.8696,C -2.6348,E1 24.9355,E2 -516.4737} C_DIS
LIN {X -18.4736,Y -37.8502,Z 61,A -122.9553,B 24.8693,C -2.6384,E1 24.9283,E2 -513.625} C_DIS
LIN {X -20.3085,Y -36.8982,Z 61,A -125.7922,B 24.869,C -2.6417,E1 24.9213,E2 -510.788} C_DIS
LIN {X -22.0545,Y -35.8816,Z 61,A -128.5497,B 24.8686,C -2.6455,E1 24.9147,E2 -508.031} C_DIS
LIN {X -23.8274,Y -34.7299,Z 61,A -131.4203,B 24.8681,C -2.65,E1 24.9081,E2 -505.1617} C_DIS
LIN {X -25.5028,Y -33.5189,Z 61,A -134.208,B 24.8676,C -2.655,E1 24.9018,E2 -502.3762} C_DIS
LIN {X -27.1168,Y -32.2272,Z 61,A -137.0679,B 24.8672,C -2.6595,E1 24.8956,E2 -499.5162} C_DIS
LIN {X -28.6308,Y -30.8896,Z 61,A -139.8628,B 24.8667,C -2.6643,E1 24.8898,E2 -496.7214} C_DIS
LIN {X -30.145,Y -29.4141,Z 61,A -142.7351,B 24.8661,C -2.6703,E1 24.8842,E2 -493.8512} C_DIS
LIN {X -31.5207,Y -27.9345,Z 61,A -145.4977,B 24.8655,C -2.6761,E1 24.879,E2 -491.0902} C_DIS
LIN {X -32.883,Y -26.3177,Z 61,A -148.3891,B 24.8649,C -2.6824,E1 24.8739,E2 -488.2007} C_DIS
LIN {X -34.107,Y -24.7104,Z 61,A -151.1529,B 24.8642,C -2.6888,E1 24.8693,E2 -485.4388} C_DIS
LIN {X -35.2136,Y -23.1054,Z 61,A -153.8975,B 24.8637,C -2.6943,E1 24.865,E2 -482.6936} C_DIS
LIN {X -36.3648,Y -21.2484,Z 61,A -156.8108,B 24.8628,C -2.7026,E1 24.8608,E2 -479.7852} C_DIS
LIN {X -37.3636,Y -19.4385,Z 61,A -159.6582,B 24.8621,C -2.7097,E1 24.857,E2 -476.9397} C_DIS
LIN {X -38.2922,Y -17.5391,Z 61,A -162.7325,B 24.8615,C -2.7153,E1 24.8534,E2 -473.8621} C_DIS
LIN {X -39.2785,Y -15.2017,Z 61,A -166.0094,B 24.8603,C -2.727,E1 24.8499,E2 -470.5949} C_DIS
LIN {X -39.9921,Y -13.2116,Z 61,A -168.8888,B 24.8595,C -2.7353,E1 24.8473,E2 -467.7189} C_DIS
LIN {X -40.5794,Y -11.2786,Z 61,A -171.6902,B 24.8587,C -2.7428,E1 24.8451,E2 -464.9192} C_DIS
LIN {X -41.0945,Y -9.2281,Z 61,A -174.5525,B 24.8578,C -2.7516,E1 24.8433,E2 -462.0611} C_DIS
LIN {X -41.4895,Y -7.2468,Z 61,A -177.3543,B 24.857,C -2.7593,E1 24.8419,E2 -459.2613} C_DIS
LIN {X -41.8011,Y -5.1557,Z 61,A 179.7664,B 24.8561,C -2.7681,E1 24.8408,E2 -456.3859} C_DIS
LIN {X -42.0037,Y -3.0984,Z 61,A 176.95,B 24.8552,C -2.7768,E1 24.8401,E2 -453.5733} C_DIS
LIN {X -42.1073,Y -0.9172,Z 61,A 173.7961,B 24.8544,C -2.7841,E1 24.8398,E2 -450.4179} C_DIS
LIN {X -42.0908,Y 1.5033,Z 61,A 170.6064,B 24.8532,C -2.7955,E1 24.84,E2 -447.2363} C_DIS
LIN {X -41.9663,Y 3.5668,Z 61,A 167.7911,B 24.8523,C -2.8043,E1 24.8405,E2 -444.4251} C_DIS
LIN {X -41.7407,Y 5.6217,Z 61,A 164.9763,B 24.8513,C -2.8131,E1 24.8415,E2 -441.6145} C_DIS
LIN {X -41.4063,Y 7.7092,Z 61,A 162.0608,B 24.8504,C -2.8216,E1 24.8429,E2 -438.7022} C_DIS
LIN {X -40.9887,Y 9.6859,Z 61,A 159.2926,B 24.8495,C -2.8299,E1 24.8445,E2 -435.9375} C_DIS
LIN {X -40.4513,Y 11.7307,Z 61,A 156.3957,B 24.8486,C -2.8385,E1 24.8467,E2 -433.0444} C_DIS
LIN {X -39.8114,Y 13.7457,Z 61,A 153.3163,B 24.8479,C -2.845,E1 24.8494,E2 -429.963} C_DIS
LIN {X -38.9118,Y 16.1178,Z 61,A 150.0628,B 24.8466,C -2.8575,E1 24.8527,E2 -426.7211} C_DIS
LIN {X -38.0939,Y 17.9651,Z 61,A 147.2385,B 24.8458,C -2.8647,E1 24.856,E2 -423.8986} C_DIS
LIN {X -37.1665,Y 19.8127,Z 61,A 144.4252,B 24.8449,C -2.8728,E1 24.8596,E2 -421.0895} C_DIS
LIN {X -36.1496,Y 21.6125,Z 61,A 141.6147,B 24.8441,C -2.8807,E1 24.8635,E2 -418.2834} C_DIS
LIN {X -35.0197,Y 23.3994,Z 61,A 138.716,B 24.8433,C -2.8883,E1 24.8679,E2 -415.3883} C_DIS
LIN {X -33.8294,Y 25.0896,Z 61,A 135.929,B 24.8424,C -2.896,E1 24.8725,E2 -412.6062} C_DIS
LIN {X -32.5871,Y 26.6828,Z 61,A 133.0873,B 24.8418,C -2.902,E1 24.8774,E2 -409.7655} C_DIS
LIN {X -31.2073,Y 28.2846,Z 61,A 130.2283,B 24.841,C -2.9094,E1 24.8827,E2 -406.9111} C_DIS
LIN {X -29.8148,Y 29.7484,Z 61,A 127.4307,B 24.8403,C -2.9153,E1 24.8882,E2 -404.1158} C_DIS
LIN {X -28.2846,Y 31.2073,Z 61,A 124.5729,B 24.8396,C -2.9221,E1 24.894,E2 -401.2626} C_DIS
LIN {X -26.7554,Y 32.5275,Z 61,A 121.7943,B 24.8389,C -2.9277,E1 24.8999,E2 -398.4867} C_DIS
LIN {X -25.1271,Y 33.8012,Z 61,A 118.9507,B 24.8383,C -2.9331,E1 24.9062,E2 -395.6456} C_DIS
LIN {X -23.4933,Y 34.9562,Z 61,A 116.1854,B 24.8378,C -2.9378,E1 24.9126,E2 -392.8823} C_DIS
LIN {X -21.6529,Y 36.1257,Z 61,A 113.2713,B 24.8371,C -2.9438,E1 24.9195,E2 -389.9735} C_DIS
LIN {X -19.8955,Y 37.1222,Z 61,A 110.4781,B 24.8367,C -2.9479,E1 24.9263,E2 -387.1819} C_DIS
LIN {X -18.05,Y 38.0537,Z 61,A 107.6555,B 24.8362,C -2.9521,E1 24.9334,E2 -384.362} C_DIS
LIN {X -16.1178,Y 38.9118,Z 61,A 104.8037,B 24.8357,C -2.9565,E1 24.9407,E2 -381.5141} C_DIS
LIN {X -14.2332,Y 39.6397,Z 61,A 102.013,B 24.8354,C -2.9595,E1 24.948,E2 -378.7246} C_DIS
LIN {X -12.271,Y 40.2904,Z 61,A 99.211,B 24.835,C -2.9628,E1 24.9554,E2 -375.9255} C_DIS
LIN {X -10.2338,Y 40.8556,Z 61,A 96.3279,B 24.8347,C -2.9655,E1 24.9632,E2 -373.0446} C_DIS
LIN {X -8.2628,Y 41.2991,Z 61,A 93.574,B 24.8345,C -2.9678,E1 24.9707,E2 -370.2928} C_DIS
LIN {X -6.18,Y 41.662,Z 61,A 90.6929,B 24.8343,C -2.9697,E1 24.9787,E2 -367.4136} C_DIS
LIN {X -4.1283,Y 41.915,Z 61,A 87.8769,B 24.8341,C -2.9711,E1 24.9865,E2 -364.5993} C_DIS
LIN {X -2.1135,Y 42.0645,Z 61,A 85.1085,B 24.8341,C -2.9719,E1 24.9942,E2 -361.8319} C_DIS
LIN {X -0.047,Y 42.1176,Z 61,A 82.3119,B 24.8339,C -2.9728,E1 25.002,E2 -359.0373} C_DIS
LIN {X 2.0197,Y 42.0691,Z 61,A 79.4813,B 24.8339,C -2.9728,E1 25.0099,E2 -356.2073} C_DIS
LIN {X 4.1283,Y 41.915,Z 61,A 76.6229,B 24.8339,C -2.9728,E1 25.0178,E2 -353.3506} C_DIS
LIN {X 6.18,Y 41.662,Z 61,A 73.812,B 24.8339,C -2.9722,E1 25.0256,E2 -350.5406} C_DIS
LIN {X 8.1707,Y 41.3175,Z 61,A 71.0483,B 24.8341,C -2.9709,E1 25.0332,E2 -347.777} C_DIS
LIN {X 10.2338,Y 40.8556,Z 61,A 68.2092,B 24.8342,C -2.9699,E1 25.0409,E2 -344.9396} C_DIS
LIN {X 12.2262,Y 40.3043,Z 61,A 65.4009,B 24.8344,C -2.9681,E1 25.0484,E2 -342.1316} C_DIS
LIN {X 14.1891,Y 39.6558,Z 61,A 62.5941,B 24.8347,C -2.9658,E1 25.0558,E2 -339.3249} C_DIS
LIN {X 16.0743,Y 38.9295,Z 61,A 59.8518,B 24.835,C -2.9632,E1 25.063,E2 -336.5826} C_DIS
LIN {X 17.9651,Y 38.0939,Z 61,A 57.0299,B 24.8354,C -2.9599,E1 25.0701,E2 -333.76} C_DIS
LIN {X 19.8542,Y 37.1446,Z 61,A 54.162,B 24.8357,C -2.9564,E1 25.0772,E2 -330.8917} C_DIS
LIN {X 21.6529,Y 36.1257,Z 61,A 51.3586,B 24.8362,C -2.9526,E1 25.084,E2 -328.0877} C_DIS
LIN {X 23.3994,Y 35.0197,Z 61,A 48.556,B 24.8366,C -2.9484,E1 25.0906,E2 -325.2843} C_DIS
LIN {X 25.0517,Y 33.8571,Z 61,A 45.8179,B 24.8371,C -2.944,E1 25.0968,E2 -322.5454} C_DIS
LIN {X 26.6828,Y 32.5871,Z 61,A 43.0034,B 24.8377,C -2.9389,E1 25.1029,E2 -319.7293} C_DIS
LIN {X 28.2496,Y 31.2386,Z 61,A 40.2346,B 24.8382,C -2.9342,E1 25.1087,E2 -316.9604} C_DIS
LIN {X 29.7818,Y 29.7818,Z 61,A 37.3758,B 24.8388,C -2.9286,E1 25.1144,E2 -314.1003} C_DIS
LIN {X 31.2073,Y 28.2846,Z 61,A 34.5717,B 24.8395,C -2.9226,E1 25.1198,E2 -311.2944} C_DIS
LIN {X 32.5575,Y 26.7193,Z 61,A 31.7577,B 24.8402,C -2.9162,E1 25.1248,E2 -308.478} C_DIS
LIN {X 33.7028,Y 25.2581,Z 61,A 29.1415,B 24.841,C -2.9088,E1 25.1293,E2 -305.8566} C_DIS
LIN {X 35.0197,Y 23.3994,Z 61,A 26.1638,B 24.8416,C -2.9031,E1 25.134,E2 -302.8802} C_DIS
LIN {X 36.1013,Y 21.693,Z 61,A 23.4138,B 24.8424,C -2.8961,E1 25.138,E2 -300.1275} C_DIS
LIN {X 37.1222,Y 19.8955,Z 61,A 20.6856,B 24.8431,C -2.8901,E1 25.1417,E2 -297.3993} C_DIS
LIN {X 38.0537,Y 18.05,Z 61,A 17.841,B 24.844,C -2.8818,E1 25.1452,E2 -294.5504} C_DIS
LIN {X 38.8936,Y 16.1611,Z 61,A 15.0464,B 24.8448,C -2.8743,E1 25.1483,E2 -291.7532} C_DIS
LIN {X 39.6397,Y 14.2332,Z 61,A 12.2944,B 24.8455,C -2.8673,E1 25.151,E2 -288.9999} C_DIS
LIN {X 40.3043,Y 12.2262,Z 61,A 9.4114,B 24.8465,C -2.8587,E1 25.1535,E2 -286.1131} C_DIS
LIN {X 40.8556,Y 10.2338,Z 61,A 6.6019,B 24.8474,C -2.8504,E1 25.1555,E2 -283.3001} C_DIS
LIN {X 41.3086,Y 8.2168,Z 61,A 3.8586,B 24.8481,C -2.8431,E1 25.1571,E2 -280.5554} C_DIS
LIN {X 41.6548,Y 6.2264,Z 61,A 1.0621,B 24.8491,C -2.8338,E1 25.1583,E2 -277.7535} C_DIS
LIN {X 41.915,Y 4.1283,Z 61,A -1.7766,B 24.85,C -2.8256,E1 25.1592,E2 -274.912} C_DIS
LIN {X 42.0671,Y 2.0666,Z 61,A -4.7478,B 24.8512,C -2.8141,E1 25.1597,E2 -271.9313} C_DIS
LIN {X 42.1147,Y -0.5169,Z 61,A -7.7214,B 24.8514,C -2.8124,E1 25.1597,E2 -268.9714} C_DIS
LIN {X 42.0691,Y -2.0197,Z 61,A -10.1077,B 24.8527,C -2.8001,E1 25.1595,E2 -266.5702} C_DIS
LIN {X 41.915,Y -4.1283,Z 61,A -12.946,B 24.8536,C -2.7917,E1 25.1588,E2 -263.7289} C_DIS
LIN {X 41.6686,Y -6.1335,Z 61,A -15.6922,B 24.8545,C -2.7831,E1 25.1578,E2 -260.9786} C_DIS
LIN {X 41.3175,Y -8.1707,Z 61,A -18.4847,B 24.8554,C -2.7747,E1 25.1564,E2 -258.1825} C_DIS
LIN {X 40.8556,Y -10.2338,Z 61,A -21.3071,B 24.8562,C -2.7667,E1 25.1546,E2 -255.3575} C_DIS
LIN {X 40.3043,Y -12.2262,Z 61,A -24.1001,B 24.8571,C -2.7584,E1 25.1524,E2 -252.5608} C_DIS
LIN {X 39.7271,Y -13.9859,Z 61,A -26.7039,B 24.858,C -2.7493,E1 25.15,E2 -249.9502} C_DIS
LIN {X 38.9295,Y -16.0743,Z 61,A -29.7003,B 24.8589,C -2.7409,E1 25.1469,E2 -246.9506} C_DIS
LIN {X 37.9549,Y -18.2557,Z 61,A -32.9714,B 24.8599,C -2.7311,E1 25.1431,E2 -243.6738} C_DIS
LIN {X 36.8982,Y -20.3085,Z 61,A -35.9882,B 24.8606,C -2.7241,E1 25.1391,E2 -240.6564} C_DIS
LIN {X 35.8816,Y -22.0545,Z 61,A -38.7192,B 24.8614,C -2.7167,E1 25.1352,E2 -237.9219} C_DIS
LIN {X 34.7299,Y -23.8274,Z 61,A -41.5617,B 24.8621,C -2.7094,E1 25.1308,E2 -235.0763} C_DIS
LIN {X 33.5189,Y -25.5028,Z 61,A -44.3732,B 24.8629,C -2.702,E1 25.1261,E2 -232.2607} C_DIS
LIN {X 32.2272,Y -27.1168,Z 61,A -47.1529,B 24.8636,C -2.6953,E1 25.1212,E2 -229.4779} C_DIS
LIN {X 30.8896,Y -28.6308,Z 61,A -49.9196,B 24.8643,C -2.6882,E1 25.116,E2 -226.7067} C_DIS
LIN {X 29.4141,Y -30.145,Z 61,A -52.7628,B 24.8649,C -2.6819,E1 25.1104,E2 -223.8607} C_DIS
LIN {X 27.9345,Y -31.5207,Z 61,A -55.4973,B 24.8655,C -2.6759,E1 25.1047,E2 -221.123} C_DIS
LIN {X 26.3177,Y -32.883,Z 61,A -58.3475,B 24.8661,C -2.6701,E1 25.0986,E2 -218.2698} C_DIS
LIN {X 24.729,Y -34.0934,Z 61,A -61.0731,B 24.8667,C -2.6644,E1 25.0925,E2 -215.5404} C_DIS
LIN {X 22.9679,Y -35.3042,Z 61,A -63.9587,B 24.8672,C -2.6591,E1 25.0858,E2 -212.652} C_DIS
LIN {X 21.2484,Y -36.3648,Z 61,A -66.6958,B 24.8677,C -2.6543,E1 25.0792,E2 -209.912} C_DIS
LIN {X 19.4385,Y -37.3636,Z 61,A -69.5149,B 24.8682,C -2.6494,E1 25.0723,E2 -207.0895} C_DIS
LIN {X 17.5391,Y -38.2922,Z 61,A -72.3475,B 24.8686,C -2.6457,E1 25.0651,E2 -204.2553} C_DIS
LIN {X 15.6391,Y -39.1067,Z 61,A -75.167,B 24.869,C -2.6416,E1 25.0578,E2 -201.4327} C_DIS
LIN {X 13.7457,Y -39.8114,Z 61,A -77.9251,B 24.8693,C -2.6379,E1 25.0506,E2 -198.6715} C_DIS
LIN {X 11.7757,Y -40.4379,Z 61,A -80.7303,B 24.8696,C -2.6349,E1 25.0431,E2 -195.864} C_DIS
LIN {X 9.7773,Y -40.967,Z 61,A -83.5189,B 24.8699,C -2.6324,E1 25.0355,E2 -193.0738} C_DIS
LIN {X 7.7092,Y -41.4063,Z 61,A -86.3735,B 24.8701,C -2.6303,E1 25.0277,E2 -190.2177} C_DIS
LIN {X 5.6683,Y -41.7347,Z 61,A -89.1815,B 24.8703,C -2.6285,E1 25.0199,E2 -187.4079} C_DIS
LIN {X 3.6604,Y -41.9582,Z 61,A -91.9605,B 24.8705,C -2.6266,E1 25.0122,E2 -184.6261} C_DIS
LIN {X 1.3169,Y -42.0965,Z 61,A -95.2686,B 24.8707,C -2.6237,E1 25.003,E2 -181.3122} C_DIS
LIN {X 1.3169,Y -42.0965,Z 61,A -95.2686,B 24.8707,C -2.6237,E1 25.003,E2 -181.3122} C_DIS
Enddeposition()
LIN {X 0.2041,Y -41.1313,Z 61,A -95.6909,B 24.8675,C -2.6561,E1 25.002,E2 -180.9671} C_DIS
Startdeposition()
$VEL.CP = VEL_PRINT
LIN {X 2.2031,Y -41.073,Z 61,A -92.1516,B 24.8663,C -2.6681,E1 25.012,E2 -184.5338} C_DIS
LIN {X 5.0158,Y -40.8257,Z 61,A -88.9533,B 24.8672,C -2.6594,E1 25.0208,E2 -187.7094} C_DIS
LIN {X 7.1261,Y -40.5103,Z 61,A -85.525,B 24.8663,C -2.6683,E1 25.0303,E2 -191.1554} C_DIS
LIN {X 9.5162,Y -40.0168,Z 61,A -82.0619,B 24.8659,C -2.6723,E1 25.0397,E2 -194.6235} C_DIS
LIN {X 11.9528,Y -39.3577,Z 61,A -78.5818,B 24.8656,C -2.6756,E1 25.0491,E2 -198.1055} C_DIS
LIN {X 14.2544,Y -38.5835,Z 61,A -75.2074,B 24.8651,C -2.6798,E1 25.058,E2 -201.4828} C_DIS
LIN {X 16.0004,Y -37.8924,Z 61,A -72.5369,B 24.8647,C -2.6843,E1 25.0649,E2 -204.158} C_DIS
LIN {X 18.1681,Y -36.9023,Z 61,A -69.0414,B 24.8639,C -2.6923,E1 25.0737,E2 -207.6633} C_DIS
LIN {X 20.8348,Y -35.465,Z 61,A -65.4847,B 24.8642,C -2.689,E1 25.0823,E2 -211.2016} C_DIS
LIN {X 22.6833,Y -34.312,Z 61,A -61.858,B 24.8627,C -2.7042,E1 25.0909,E2 -214.8528} C_DIS
LIN {X 24.677,Y -32.9073,Z 61,A -58.5968,B 24.8622,C -2.7089,E1 25.0982,E2 -218.1135} C_DIS
LIN {X 26.6137,Y -31.3618,Z 61,A -55.5422,B 24.8621,C -2.7099,E1 25.1048,E2 -221.1587} C_DIS
LIN {X 28.3542,Y -29.7984,Z 61,A -51.6199,B 24.8602,C -2.7283,E1 25.1129,E2 -225.1088} C_DIS
LIN {X 30.7661,Y -27.3007,Z 61,A -47.1498,B 24.8596,C -2.734,E1 25.1214,E2 -229.5728} C_DIS
LIN {X 31.8438,Y -26.0355,Z 61,A -44.3527,B 24.8582,C -2.7481,E1 25.1264,E2 -232.3902} C_DIS
LIN {X 34.1929,Y -22.8629,Z 61,A -39.4755,B 24.8577,C -2.7523,E1 25.1342,E2 -237.2536} C_DIS
LIN {X 35.3903,Y -20.9612,Z 61,A -36.3996,B 24.8569,C -2.7601,E1 25.1387,E2 -240.3324} C_DIS
LIN {X 36.4897,Y -18.9839,Z 61,A -33.337,B 24.8561,C -2.7676,E1 25.1427,E2 -243.3967} C_DIS
LIN {X 37.2828,Y -17.3734,Z 61,A -30.7849,B 24.8553,C -2.7758,E1 25.1458,E2 -245.9544} C_DIS
LIN {X 38.0735,Y -15.5647,Z 61,A -28.2012,B 24.8547,C -2.7812,E1 25.1486,E2 -248.5366} C_DIS
LIN {X 38.8428,Y -13.531,Z 61,A -25.1301,B 24.8537,C -2.791,E1 25.1516,E2 -251.6139} C_DIS
LIN {X 39.4944,Y -11.4912,Z 61,A -22.1728,B 24.8528,C -2.7997,E1 25.154,E2 -254.5748} C_DIS
LIN {X 40.058,Y -9.3385,Z 61,A -18.8508,B 24.8513,C -2.8132,E1 25.1562,E2 -257.9095} C_DIS
LIN {X 40.5327,Y -6.9994,Z 61,A -15.6298,B 24.8504,C -2.8217,E1 25.1579,E2 -261.1319} C_DIS
LIN {X 40.8659,Y -4.6724,Z 61,A -12.4715,B 24.8495,C -2.83,E1 25.159,E2 -264.2911} C_DIS
LIN {X 41.0386,Y -2.7706,Z 61,A -10.0623,B 24.8491,C -2.834,E1 25.1595,E2 -266.6955} C_DIS
LIN {X 41.1305,Y 0.2884,Z 61,A -5.5868,B 24.8473,C -2.8511,E1 25.1597,E2 -271.1847} C_DIS
LIN {X 41.0472,Y 2.6441,Z 61,A -2.1896,B 24.846,C -2.8633,E1 25.1593,E2 -274.5906} C_DIS
LIN {X 40.7907,Y 5.2877,Z 61,A 1.799,B 24.8442,C -2.8797,E1 25.158,E2 -278.5945} C_DIS
LIN {X 40.0737,Y 9.2707,Z 61,A 7.0601,B 24.843,C -2.8903,E1 25.1551,E2 -283.8499} C_DIS
LIN {X 39.5203,Y 11.4032,Z 61,A 10.356,B 24.8416,C -2.9032,E1 25.1526,E2 -287.1576} C_DIS
LIN {X 38.6987,Y 13.9385,Z 61,A 13.8162,B 24.8409,C -2.9097,E1 25.1495,E2 -290.6136} C_DIS
LIN {X 37.7666,Y 16.2958,Z 61,A 17.3164,B 24.8399,C -2.9191,E1 25.1457,E2 -294.1168} C_DIS
LIN {X 36.695,Y 18.5834,Z 61,A 20.5359,B 24.8394,C -2.9236,E1 25.1418,E2 -297.3298} C_DIS
LIN {X 35.211,Y 21.2613,Z 61,A 25.0139,B 24.8378,C -2.9384,E1 25.1356,E2 -301.8195} C_DIS
LIN {X 33.8864,Y 23.3151,Z 61,A 28.3766,B 24.8369,C -2.9461,E1 25.1304,E2 -305.1839} C_DIS
LIN {X 32.5535,Y 25.142,Z 61,A 31.8393,B 24.8355,C -2.9588,E1 25.1245,E2 -308.6602} C_DIS
LIN {X 30.6051,Y 27.4805,Z 61,A 35.6748,B 24.8352,C -2.9617,E1 25.1176,E2 -312.4851} C_DIS
LIN {X 29.0543,Y 29.1159,Z 61,A 38.7975,B 24.8344,C -2.968,E1 25.1115,E2 -315.6094} C_DIS
LIN {X 27.3042,Y 30.7629,Z 61,A 42.4225,B 24.8332,C -2.979,E1 25.104,E2 -319.2459} C_DIS
LIN {X 25.3198,Y 32.4156,Z 61,A 45.9548,B 24.8326,C -2.9845,E1 25.0963,E2 -322.7779} C_DIS
LIN {X 23.1961,Y 33.9678,Z 61,A 49.4495,B 24.8322,C -2.9878,E1 25.0883,E2 -326.2684} C_DIS
LIN {X 20.5397,Y 35.6366,Z 61,A 53.8179,B 24.8315,C -2.9941,E1 25.0779,E2 -330.6382} C_DIS
LIN {X 18.5365,Y 36.719,Z 61,A 56.9952,B 24.831,C -2.9982,E1 25.07,E2 -333.8163} C_DIS
LIN {X 16.2939,Y 37.7674,Z 61,A 60.397,B 24.8307,C -3.0013,E1 25.0613,E2 -337.2171} C_DIS
LIN {X 14.0345,Y 38.6637,Z 61,A 63.7485,B 24.8304,C -3.004,E1 25.0526,E2 -340.5677} C_DIS
LIN {X 11.6804,Y 39.4387,Z 61,A 67.1772,B 24.8301,C -3.0062,E1 25.0434,E2 -343.9954} C_DIS
LIN {X 9.2726,Y 40.0732,Z 61,A 70.7025,B 24.8298,C -3.009,E1 25.0339,E2 -347.5221} C_DIS
LIN {X 6.7571,Y 40.5732,Z 61,A 74.2311,B 24.8298,C -3.0097,E1 25.0242,E2 -351.0485} C_DIS
LIN {X 4.6563,Y 40.8675,Z 61,A 77.7106,B 24.8288,C -3.0177,E1 25.0145,E2 -354.5444} C_DIS
LIN {X 0.6903,Y 41.1263,Z 61,A 82.7126,B 24.8297,C -3.0099,E1 25.0006,E2 -359.5263} C_DIS
LIN {X -2.3898,Y 41.0627,Z 61,A 87.0761,B 24.8297,C -3.0096,E1 24.9884,E2 -363.8897} C_DIS
LIN {X -4.9438,Y 40.8342,Z 61,A 90.4594,B 24.8303,C -3.0052,E1 24.9791,E2 -367.2645} C_DIS
LIN {X -7.171,Y 40.5023,Z 61,A 93.5423,B 24.8306,C -3.0023,E1 24.9706,E2 -370.3435} C_DIS
LIN {X -10.428,Y 39.7887,Z 61,A 98.4442,B 24.8306,C -3.0015,E1 24.9572,E2 -375.2498} C_DIS
LIN {X -12.7212,Y 39.1155,Z 61,A 101.6441,B 24.8313,C -2.9962,E1 24.9487,E2 -378.4425} C_DIS
LIN {X -14.7327,Y 38.4034,Z 61,A 104.5955,B 24.8317,C -2.9921,E1 24.941,E2 -381.3904} C_DIS
LIN {X -16.5532,Y 37.6544,Z 61,A 107.0533,B 24.8326,C -2.9848,E1 24.9347,E2 -383.8362} C_DIS
LIN {X -18.3171,Y 36.8284,Z 61,A 110.4098,B 24.8321,C -2.9885,E1 24.9262,E2 -387.2105} C_DIS
LIN {X -21.0724,Y 35.3245,Z 61,A 114.2587,B 24.8337,C -2.9747,E1 24.9169,E2 -391.0375} C_DIS
LIN {X -23.646,Y 33.6564,Z 61,A 118.9414,B 24.8341,C -2.9715,E1 24.906,E2 -395.728} C_DIS
LIN {X -25.6226,Y 32.1769,Z 61,A 121.9967,B 24.8354,C -2.9599,E1 24.8993,E2 -398.7666} C_DIS
LIN {X -27.52,Y 30.5698,Z 61,A 125.7311,B 24.8359,C -2.9554,E1 24.8914,E2 -402.5051} C_DIS
LIN {X -29.2032,Y 28.9659,Z 61,A 129.0872,B 24.8365,C -2.9492,E1 24.8847,E2 -405.8604} C_DIS
LIN {X -31.1124,Y 26.9054,Z 61,A 132.8857,B 24.8378,C -2.9383,E1 24.8776,E2 -409.6498} C_DIS
LIN {X -32.7477,Y 24.8895,Z 61,A 137.2719,B 24.8378,C -2.9377,E1 24.8701,E2 -414.0553} C_DIS
LIN {X -35.0996,Y 21.4446,Z 61,A 142.1135,B 24.8408,C -2.911,E1 24.8627,E2 -418.8572} C_DIS
LIN {X -36.1103,Y 19.6952,Z 61,A 145.4061,B 24.8411,C -2.9084,E1 24.8582,E2 -422.1608} C_DIS
LIN {X -37.2852,Y 17.3682,Z 61,A 148.9843,B 24.8423,C -2.8972,E1 24.8538,E2 -425.7318} C_DIS
LIN {X -38.247,Y 15.1336,Z 61,A 152.3027,B 24.8435,C -2.8864,E1 24.8503,E2 -429.0426} C_DIS
LIN {X -38.9253,Y 13.2926,Z 61,A 155.5508,B 24.8437,C -2.8838,E1 24.8473,E2 -432.303} C_DIS
LIN {X -39.7836,Y 10.4477,Z 61,A 159.4132,B 24.8455,C -2.8681,E1 24.8444,E2 -436.1502} C_DIS
LIN {X -40.3625,Y 7.9207,Z 61,A 162.9938,B 24.8467,C -2.8565,E1 24.8423,E2 -439.7242} C_DIS
LIN {X -40.7753,Y 5.4069,Z 61,A 166.5996,B 24.8478,C -2.8461,E1 24.8409,E2 -443.3264} C_DIS
LIN {X -41.0344,Y 2.8331,Z 61,A 170.0558,B 24.8492,C -2.8332,E1 24.84,E2 -446.7726} C_DIS
LIN {X -41.12,Y 1.0204,Z 61,A 172.8131,B 24.8498,C -2.8277,E1 24.8398,E2 -449.5334} C_DIS
LIN {X -41.1052,Y -1.5057,Z 61,A 176.3374,B 24.8509,C -2.8168,E1 24.84,E2 -453.0528} C_DIS
LIN {X -40.9393,Y -3.9822,Z 61,A 179.7279,B 24.8522,C -2.8054,E1 24.8408,E2 -456.4362} C_DIS
LIN {X -40.6373,Y -6.3609,Z 61,A -176.9192,B 24.8532,C -2.7953,E1 24.8421,E2 -459.7849} C_DIS
LIN {X -40.1488,Y -8.9409,Z 61,A -173.022,B 24.8541,C -2.7868,E1 24.8443,E2 -463.685} C_DIS
LIN {X -39.5592,Y -11.2656,Z 61,A -169.8903,B 24.8554,C -2.7746,E1 24.8466,E2 -466.8057} C_DIS
LIN {X -38.8852,Y -13.4101,Z 61,A -166.7508,B 24.8563,C -2.7656,E1 24.8493,E2 -469.9415} C_DIS
LIN {X -38.0498,Y -15.6227,Z 61,A -163.4384,B 24.8573,C -2.7565,E1 24.8527,E2 -473.2507} C_DIS
LIN {X -37.269,Y -17.403,Z 61,A -160.8183,B 24.8582,C -2.748,E1 24.8557,E2 -475.8649} C_DIS
LIN {X -36.4346,Y -19.0885,Z 61,A -158.1049,B 24.8588,C -2.742,E1 24.8592,E2 -478.5785} C_DIS
LIN {X -35.3823,Y -20.9747,Z 61,A -154.7158,B 24.8591,C -2.7386,E1 24.8639,E2 -481.977} C_DIS
LIN {X -34.3752,Y -22.5875,Z 61,A -151.3643,B 24.859,C -2.7402,E1 24.8691,E2 -485.3491} C_DIS
LIN {X -32.2544,Y -25.5245,Z 61,A -147.2986,B 24.8614,C -2.7167,E1 24.8759,E2 -489.3781} C_DIS
LIN {X -30.7645,Y -27.3024,Z 61,A -143.9603,B 24.862,C -2.7107,E1 24.882,E2 -492.7174} C_DIS
LIN {X -29.0356,Y -29.1343,Z 61,A -140.4851,B 24.8628,C -2.703,E1 24.8888,E2 -496.189} C_DIS
LIN {X -27.5913,Y -30.5059,Z 61,A -137.8694,B 24.8635,C -2.6956,E1 24.8941,E2 -498.7977} C_DIS
LIN {X -26.2104,Y -31.6997,Z 61,A -134.8508,B 24.8635,C -2.6968,E1 24.9006,E2 -501.8307} C_DIS
LIN {X -24.6498,Y -32.9278,Z 61,A -132.0765,B 24.8639,C -2.6922,E1 24.9068,E2 -504.6039} C_DIS
LIN {X -22.2542,Y -34.5919,Z 61,A -128.2465,B 24.8648,C -2.6829,E1 24.9157,E2 -508.4245} C_DIS
LIN {X -20.1357,Y -35.8665,Z 61,A -124.8194,B 24.8653,C -2.6779,E1 24.9239,E2 -511.85} C_DIS
LIN {X -18.0118,Y -36.9793,Z 61,A -121.4499,B 24.8657,C -2.6743,E1 24.9323,E2 -515.2197} C_DIS
LIN {X -15.8297,Y -37.9643,Z 61,A -118.0581,B 24.866,C -2.6716,E1 24.941,E2 -518.6131} C_DIS
LIN {X -13.5725,Y -38.8283,Z 61,A -114.754,B 24.8663,C -2.6678,E1 24.9497,E2 -521.9149} C_DIS
LIN {X -11.4893,Y -39.4954,Z 61,A -111.5866,B 24.8663,C -2.6673,E1 24.9582,E2 -525.0866} C_DIS
LIN {X -8.9811,Y -40.1402,Z 61,A -108.1189,B 24.8668,C -2.6636,E1 24.9676,E2 -528.5501} C_DIS
LIN {X -6.3748,Y -40.6351,Z 61,A -103.8616,B 24.8661,C -2.6703,E1 24.9793,E2 -532.8275} C_DIS
LIN {X -3.1394,Y -41.0123,Z 61,A -100.1615,B 24.8673,C -2.6581,E1 24.9895,E2 -536.5006} C_DIS
LIN {X -1.1004,Y -41.1176,Z 61,A -96.9664,B 24.8668,C -2.6634,E1 24.9985,E2 -539.7089} C_DIS
LIN {X -1.1004,Y -41.1176,Z 61,A -96.9664,B 24.8668,C -2.6634,E1 24.9985,E2 -539.7089} C_DIS
Enddeposition()
LIN {X 0.2062,Y -40.1412,Z 61,A -96.4339,B 24.8668,C -2.6627,E1 25,E2 -540.2397} C_DIS
Startdeposition()
$VEL.CP = VEL_PRINT
LIN {X -2.4537,Y -40.0725,Z 61,A -100.2083,B 24.8668,C -2.6625,E1 24.9894,E2 -536.4641} C_DIS
LIN {X -3.8295,Y -39.9642,Z 61,A -102.9268,B 24.8679,C -2.6526,E1 24.9818,E2 -533.7207} C_DIS
LIN {X -7.0008,Y -39.5319,Z 61,A -106.8017,B 24.8669,C -2.6628,E1 24.9712,E2 -529.8669} C_DIS
LIN {X -8.7341,Y -39.1859,Z 61,A -109.5943,B 24.8671,C -2.6603,E1 24.9635,E2 -527.065} C_DIS
LIN {X -10.7789,Y -38.6734,Z 61,A -112.7627,B 24.8671,C -2.66,E1 24.9549,E2 -523.8912} C_DIS
LIN {X -12.8301,Y -38.0417,Z 61,A -115.8648,B 24.8669,C -2.6619,E1 24.9467,E2 -520.7878} C_DIS
LIN {X -15.9061,Y -36.8619,Z 61,A -120.5591,B 24.8665,C -2.6664,E1 24.9345,E2 -516.0941} C_DIS
LIN {X -18.0716,Y -35.8504,Z 61,A -123.9182,B 24.866,C -2.6711,E1 24.9261,E2 -512.7373} C_DIS
LIN {X -20.0839,Y -34.7625,Z 61,A -127.1621,B 24.8656,C -2.6757,E1 24.9182,E2 -509.495} C_DIS
LIN {X -21.9149,Y -33.6385,Z 61,A -130.0057,B 24.8648,C -2.6828,E1 24.9115,E2 -506.6595} C_DIS
LIN {X -23.8215,Y -32.316,Z 61,A -133.187,B 24.8641,C -2.6898,E1 24.9043,E2 -503.4837} C_DIS
LIN {X -24.9634,Y -31.4421,Z 61,A -135.8828,B 24.8645,C -2.6859,E1 24.8983,E2 -500.7688} C_DIS
LIN {X -27.0549,Y -29.6619,Z 61,A -139.8445,B 24.8638,C -2.6929,E1 24.89,E2 -496.808} C_DIS
LIN {X -29.3908,Y -27.3496,Z 61,A -143.8258,B 24.862,C -2.7106,E1 24.8823,E2 -492.8522} C_DIS
LIN {X -30.8913,Y -25.6419,Z 61,A -147.8122,B 24.8621,C -2.7096,E1 24.875,E2 -488.8452} C_DIS
LIN {X -32.5344,Y -23.5219,Z 61,A -151.5534,B 24.8611,C -2.7197,E1 24.8687,E2 -485.1101} C_DIS
LIN {X -33.9048,Y -21.5011,Z 61,A -155.3732,B 24.8606,C -2.7248,E1 24.8629,E2 -481.2832} C_DIS
LIN {X -35.7343,Y -18.2987,Z 61,A -160.6901,B 24.8592,C -2.7382,E1 24.8558,E2 -475.9703} C_DIS
LIN {X -37.3302,Y -14.7733,Z 61,A -165.8351,B 24.8572,C -2.7575,E1 24.8502,E2 -470.8432} C_DIS
LIN {X -38.1358,Y -12.5494,Z 61,A -169.0135,B 24.8559,C -2.7693,E1 24.8473,E2 -467.6749} C_DIS
LIN {X -38.5663,Y -11.1566,Z 61,A -171.272,B 24.8555,C -2.7736,E1 24.8455,E2 -465.4136} C_DIS
LIN {X -39.099,Y -9.1135,Z 61,A -174.1428,B 24.8544,C -2.7841,E1 24.8436,E2 -462.551} C_DIS
LIN {X -39.5714,Y -6.7759,Z 61,A -177.829,B 24.8536,C -2.7915,E1 24.8417,E2 -458.8608} C_DIS
LIN {X -39.9184,Y -4.2798,Z 61,A 178.6265,B 24.8524,C -2.8031,E1 24.8405,E2 -455.3229} C_DIS
LIN {X -40.0704,Y -2.4894,Z 61,A 175.8928,B 24.8517,C -2.8094,E1 24.8399,E2 -452.5877} C_DIS
LIN {X -40.1455,Y 0.2804,Z 61,A 171.5117,B 24.8509,C -2.8175,E1 24.8399,E2 -448.1996} C_DIS
LIN {X -39.9934,Y 3.5132,Z 61,A 167.421,B 24.8488,C -2.8372,E1 24.8406,E2 -444.1316} C_DIS
LIN {X -39.7462,Y 5.6589,Z 61,A 164.3991,B 24.8477,C -2.8475,E1 24.8417,E2 -441.1162} C_DIS
LIN {X -39.3956,Y 7.7323,Z 61,A 161.3955,B 24.8467,C -2.8568,E1 24.8432,E2 -438.1171} C_DIS
LIN {X -38.9421,Y 9.7647,Z 61,A 158.2915,B 24.8458,C -2.8646,E1 24.8452,E2 -435.0137} C_DIS
LIN {X -38.4869,Y 11.4256,Z 61,A 155.3905,B 24.8455,C -2.8677,E1 24.8475,E2 -432.1032} C_DIS
LIN {X -37.1814,Y 15.1436,Z 61,A 150.1422,B 24.8432,C -2.8884,E1 24.8526,E2 -426.8748} C_DIS
LIN {X -36.1559,Y 17.4511,Z 61,A 146.5665,B 24.8421,C -2.8992,E1 24.8567,E2 -423.3055} C_DIS
LIN {X -35.1949,Y 19.3168,Z 61,A 143.6203,B 24.8411,C -2.9083,E1 24.8606,E2 -420.3653} C_DIS
LIN {X -34.2482,Y 20.9488,Z 61,A 141.03,B 24.8401,C -2.9169,E1 24.8643,E2 -417.7822} C_DIS
LIN {X -32.9949,Y 22.8718,Z 61,A 137.0188,B 24.84,C -2.918,E1 24.8706,E2 -413.7538} C_DIS
LIN {X -31.2373,Y 25.2194,Z 61,A 133.1752,B 24.8384,C -2.9324,E1 24.8771,E2 -409.9266} C_DIS
LIN {X -29.5965,Y 27.1262,Z 61,A 129.4702,B 24.8376,C -2.9401,E1 24.884,E2 -406.2232} C_DIS
LIN {X -27.1692,Y 29.557,Z 61,A 124.4624,B 24.8364,C -2.9503,E1 24.8941,E2 -401.219} C_DIS
LIN {X -25.5414,Y 30.9747,Z 61,A 121.6939,B 24.8353,C -2.9604,E1 24.9,E2 -398.464} C_DIS
LIN {X -23.6614,Y 32.4334,Z 61,A 118.845,B 24.8338,C -2.9735,E1 24.9062,E2 -395.6361} C_DIS
LIN {X -21.9123,Y 33.6393,Z 61,A 115.5742,B 24.8335,C -2.9766,E1 24.9138,E2 -392.3617} C_DIS
LIN {X -20.7738,Y 34.3547,Z 61,A 113.2911,B 24.8335,C -2.9759,E1 24.9192,E2 -390.0698} C_DIS
LIN {X -18.6591,Y 35.5475,Z 61,A 110.2906,B 24.8323,C -2.9871,E1 24.9265,E2 -387.0874} C_DIS
LIN {X -16.1585,Y 36.7519,Z 61,A 105.8035,B 24.8323,C -2.9868,E1 24.9379,E2 -382.5884} C_DIS
LIN {X -14.0815,Y 37.5968,Z 61,A 102.6546,B 24.8318,C -2.9917,E1 24.9461,E2 -379.4443} C_DIS
LIN {X -11.5946,Y 38.4367,Z 61,A 98.3993,B 24.832,C -2.9898,E1 24.9574,E2 -375.1769} C_DIS
LIN {X -7.8254,Y 39.3777,Z 61,A 93.3179,B 24.8308,C -3.0004,E1 24.9712,E2 -370.1142} C_DIS
LIN {X -5.6937,Y 39.7413,Z 61,A 90.2211,B 24.8306,C -3.0024,E1 24.9798,E2 -367.0194} C_DIS
LIN {X -3.4247,Y 40.0013,Z 61,A 87.2353,B 24.83,C -3.0075,E1 24.988,E2 -364.044} C_DIS
LIN {X -1.519,Y 40.118,Z 61,A 84.579,B 24.8298,C -3.0094,E1 24.9954,E2 -361.3915} C_DIS
LIN {X -0.1811,Y 40.1467,Z 61,A 82.4885,B 24.83,C -3.0075,E1 25.0013,E2 -359.2963} C_DIS
LIN {X 1.5565,Y 40.1172,Z 61,A 79.9212,B 24.83,C -3.0066,E1 25.0084,E2 -356.7275} C_DIS
LIN {X 3.5742,Y 39.9877,Z 61,A 76.4685,B 24.831,C -2.9989,E1 25.0181,E2 -353.2582} C_DIS
LIN {X 6.6403,Y 39.5941,Z 61,A 72.5443,B 24.8304,C -3.0043,E1 25.0289,E2 -349.3505} C_DIS
LIN {X 9.0083,Y 39.1233,Z 61,A 69.4301,B 24.83,C -3.0073,E1 25.0374,E2 -346.2474} C_DIS
LIN {X 11.0886,Y 38.5855,Z 61,A 65.5299,B 24.8316,C -2.9937,E1 25.0479,E2 -342.3213} C_DIS
LIN {X 13.8799,Y 37.6716,Z 61,A 61.8405,B 24.8312,C -2.9973,E1 25.0576,E2 -338.6476} C_DIS
LIN {X 16.0904,Y 36.7816,Z 61,A 58.4153,B 24.8316,C -2.9934,E1 25.0664,E2 -335.2213} C_DIS
LIN {X 18.3545,Y 35.7058,Z 61,A 54.8648,B 24.832,C -2.9895,E1 25.0753,E2 -331.671} C_DIS
LIN {X 20.3762,Y 34.5918,Z 61,A 51.565,B 24.8326,C -2.9849,E1 25.0833,E2 -328.3701} C_DIS
LIN {X 22.18,Y 33.464,Z 61,A 48.5951,B 24.833,C -2.9812,E1 25.0903,E2 -325.4011} C_DIS
LIN {X 24.1458,Y 32.0744,Z 61,A 45.1619,B 24.8336,C -2.9754,E1 25.0981,E2 -321.9665} C_DIS
LIN {X 25.9217,Y 30.6565,Z 61,A 41.6864,B 24.8347,C -2.966,E1 25.1056,E2 -318.4817} C_DIS
LIN {X 28.0018,Y 28.7701,Z 61,A 37.8595,B 24.8353,C -2.9607,E1 25.1133,E2 -314.6581} C_DIS
LIN {X 29.6218,Y 27.0986,Z 61,A 34.6597,B 24.8358,C -2.9555,E1 25.1195,E2 -311.4598} C_DIS
LIN {X 31.2146,Y 25.2475,Z 61,A 30.7055,B 24.8375,C -2.9403,E1 25.1266,E2 -307.4877} C_DIS
LIN {X 32.7082,Y 23.28,Z 61,A 27.3933,B 24.8381,C -2.9351,E1 25.132,E2 -304.1793} C_DIS
LIN {X 34.2418,Y 20.9594,Z 61,A 23.8775,B 24.8384,C -2.9323,E1 25.1373,E2 -300.6745} C_DIS
LIN {X 35.186,Y 19.3328,Z 61,A 20.515,B 24.8404,C -2.9144,E1 25.1419,E2 -297.2871} C_DIS
LIN {X 36.5483,Y 16.6138,Z 61,A 16.7882,B 24.8406,C -2.9123,E1 25.1463,E2 -293.5755} C_DIS
LIN {X 37.4554,Y 14.4546,Z 61,A 13.2902,B 24.8419,C -2.9004,E1 25.15,E2 -290.0685} C_DIS
LIN {X 38.3526,Y 11.8684,Z 61,A 9.189,B 24.8435,C -2.8858,E1 25.1536,E2 -285.9562} C_DIS
LIN {X 39.1027,Y 9.0976,Z 61,A 5.9857,B 24.8433,C -2.8883,E1 25.1558,E2 -282.7771} C_DIS
LIN {X 39.5361,Y 6.9786,Z 61,A 2.6312,B 24.8448,C -2.8745,E1 25.1576,E2 -279.4095} C_DIS
LIN {X 39.8087,Y 5.2012,Z 61,A -0.0601,B 24.8458,C -2.8645,E1 25.1587,E2 -276.7105} C_DIS
LIN {X 40.0219,Y 3.1667,Z 61,A -3.435,B 24.8476,C -2.848,E1 25.1595,E2 -273.3165} C_DIS
LIN {X 40.134,Y 1.0401,Z 61,A -6.2287,B 24.8482,C -2.8425,E1 25.1598,E2 -270.5264} C_DIS
LIN {X 40.1213,Y -1.4241,Z 61,A -9.2961,B 24.8486,C -2.839,E1 25.1596,E2 -267.4689} C_DIS
LIN {X 40.0365,Y -2.9841,Z 61,A -12.0439,B 24.8503,C -2.8233,E1 25.1591,E2 -264.7004} C_DIS
LIN {X 39.6869,Y -6.0612,Z 61,A -16.1369,B 24.8511,C -2.8149,E1 25.1576,E2 -260.6117} C_DIS
LIN {X 39.2966,Y -8.2207,Z 61,A -19.2615,B 24.8522,C -2.8053,E1 25.156,E2 -257.4824} C_DIS
LIN {X 38.8934,Y -9.9544,Z 61,A -21.5012,B 24.8525,C -2.8024,E1 25.1545,E2 -255.2489} C_DIS
LIN {X 38.364,Y -11.8316,Z 61,A -25.2563,B 24.8551,C -2.7778,E1 25.1514,E2 -251.4572} C_DIS
LIN {X 37.1202,Y -15.2938,Z 61,A -30.1533,B 24.8561,C -2.7679,E1 25.1465,E2 -246.5638} C_DIS
LIN {X 36.0877,Y -17.5929,Z 61,A -33.2991,B 24.8564,C -2.7647,E1 25.1428,E2 -243.4275} C_DIS
LIN {X 34.7324,Y -20.1362,Z 61,A -37.4214,B 24.8577,C -2.7528,E1 25.1372,E2 -239.2986} C_DIS
LIN {X 32.7638,Y -23.202,Z 61,A -42.4829,B 24.8589,C -2.7408,E1 25.1294,E2 -234.2339} C_DIS
LIN {X 31.0085,Y -25.501,Z 61,A -46.6333,B 24.8601,C -2.7297,E1 25.1223,E2 -230.0767} C_DIS
LIN {X 30.0916,Y -26.5758,Z 61,A -49.284,B 24.8616,C -2.7146,E1 25.1173,E2 -227.402} C_DIS
LIN {X 27.5705,Y -29.1832,Z 61,A -54.1955,B 24.8624,C -2.7065,E1 25.1076,E2 -222.4922} C_DIS
LIN {X 24.9397,Y -31.4607,Z 61,A -58.6821,B 24.8628,C -2.7032,E1 25.098,E2 -218.0149} C_DIS
LIN {X 23.7084,Y -32.399,Z 61,A -61.9804,B 24.8649,C -2.6819,E1 25.0905,E2 -214.6778} C_DIS
LIN {X 20.6439,Y -34.4328,Z 61,A -66.0888,B 24.8642,C -2.6895,E1 25.0809,E2 -210.6008} C_DIS
LIN {X 19.1818,Y -35.2682,Z 61,A -68.7207,B 24.8649,C -2.6819,E1 25.0744,E2 -207.9585} C_DIS
LIN {X 17.6454,Y -36.062,Z 61,A -71.6483,B 24.866,C -2.6711,E1 25.067,E2 -205.0131} C_DIS
LIN {X 14.4032,Y -37.4749,Z 61,A -76.2135,B 24.866,C -2.6711,E1 25.0553,E2 -200.4586} C_DIS
LIN {X 12.0433,Y -38.2984,Z 61,A -79.7494,B 24.8664,C -2.6673,E1 25.0459,E2 -196.9203} C_DIS
LIN {X 9.7329,Y -38.95,Z 61,A -83.2056,B 24.8668,C -2.6634,E1 25.0366,E2 -193.4602} C_DIS
LIN {X 6.6753,Y -39.5882,Z 61,A -87.8326,B 24.8674,C -2.6574,E1 25.0239,E2 -188.8243} C_DIS
LIN {X 4.4515,Y -39.9001,Z 61,A -90.5689,B 24.8669,C -2.662,E1 25.0163,E2 -186.101} C_DIS
LIN {X 2.946,Y -40.0393,Z 61,A -92.9745,B 24.8674,C -2.6575,E1 25.0096,E2 -183.686} C_DIS
LIN {X 0.6371,Y -40.1421,Z 61,A -96.4144,B 24.8677,C -2.6545,E1 25,E2 -180.2397} C_DIS
LIN {X 0.6371,Y -40.1421,Z 61,A -96.4144,B 24.8677,C -2.6545,E1 25,E2 -180.2397} C_DIS
Enddeposition()
LIN {X 0.2046,Y -39.1588,Z 61,A -96.2597,B 24.8649,C -2.6821,E1 25.0006,E2 -180.4601} C_DIS
Startdeposition()
$VEL.CP = VEL_PRINT
LIN {X 1.3377,Y -39.1394,Z 61,A -93.8488,B 24.8638,C -2.6928,E1 25.0074,E2 -182.8961} C_DIS
LIN {X 3.1696,Y -39.0336,Z 61,A -90.8808,B 24.8633,C -2.698,E1 25.0157,E2 -185.8749} C_DIS
LIN {X 4.9623,Y -38.8464,Z 61,A -87.6737,B 24.8623,C -2.7077,E1 25.0246,E2 -189.1025} C_DIS
LIN {X 8.8169,Y -38.1566,Z 61,A -82.7654,B 24.863,C -2.7006,E1 25.038,E2 -193.9882} C_DIS
LIN {X 10.4113,Y -37.7533,Z 61,A -80.1617,B 24.8625,C -2.706,E1 25.045,E2 -196.6005} C_DIS
LIN {X 12.6722,Y -37.0554,Z 61,A -76.6691,B 24.862,C -2.7105,E1 25.0543,E2 -200.0973} C_DIS
LIN {X 14.9796,Y -36.1836,Z 61,A -73.3446,B 24.862,C -2.7112,E1 25.063,E2 -203.4161} C_DIS
LIN {X 17.0376,Y -35.2617,Z 61,A -69.5212,B 24.8606,C -2.7241,E1 25.0727,E2 -207.2604} C_DIS
LIN {X 19.15,Y -34.1606,Z 61,A -66.1942,B 24.8603,C -2.7277,E1 25.0808,E2 -210.5861} C_DIS
LIN {X 21.2969,Y -32.8654,Z 61,A -62.8049,B 24.86,C -2.7302,E1 25.0889,E2 -213.9705} C_DIS
LIN {X 23.0217,Y -31.681,Z 61,A -59.7338,B 24.8594,C -2.7364,E1 25.0959,E2 -217.0458} C_DIS
LIN {X 24.5605,Y -30.5034,Z 61,A -56.9823,B 24.8589,C -2.7411,E1 25.1019,E2 -219.7982} C_DIS
LIN {X 26.0695,Y -29.2241,Z 61,A -53.9842,B 24.858,C -2.7492,E1 25.1082,E2 -222.8036} C_DIS
LIN {X 27.6927,Y -27.6915,Z 61,A -50.6245,B 24.8571,C -2.7583,E1 25.115,E2 -226.171} C_DIS
LIN {X 29.0818,Y -26.2283,Z 61,A -47.9332,B 24.8568,C -2.7614,E1 25.1201,E2 -228.8578} C_DIS
LIN {X 30.3073,Y -24.8025,Z 61,A -45.0163,B 24.8558,C -2.7711,E1 25.1253,E2 -231.7842} C_DIS
LIN {X 31.6484,Y -23.0661,Z 61,A -42.0827,B 24.8553,C -2.7751,E1 25.1302,E2 -234.7133} C_DIS
LIN {X 32.5889,Y -21.7171,Z 61,A -39.3768,B 24.8541,C -2.7865,E1 25.1345,E2 -237.4328} C_DIS
LIN {X 33.4276,Y -20.4026,Z 61,A -36.8952,B 24.8531,C -2.7961,E1 25.1381,E2 -239.9246} C_DIS
LIN {X 34.7419,Y -18.0749,Z 61,A -33.5591,B 24.8529,C -2.7979,E1 25.1426,E2 -243.2474} C_DIS
LIN {X 35.4422,Y -16.6593,Z 61,A -31.4485,B 24.8526,C -2.8014,E1 25.1451,E2 -245.3549} C_DIS
LIN {X 36.1665,Y -15.0228,Z 61,A -28.4253,B 24.8511,C -2.8158,E1 25.1485,E2 -248.3957} C_DIS
LIN {X 37.1206,Y -12.479,Z 61,A -24.2139,B 24.8494,C -2.8317,E1 25.1524,E2 -252.6211} C_DIS
LIN {X 37.6997,Y -10.6018,Z 61,A -20.9696,B 24.8478,C -2.8467,E1 25.1549,E2 -255.8823} C_DIS
LIN {X 38.5434,Y -6.9332,Z 61,A -16.3008,B 24.8474,C -2.8499,E1 25.1576,E2 -260.5314} C_DIS
LIN {X 38.8273,Y -5.1079,Z 61,A -13.3996,B 24.8461,C -2.8616,E1 25.1587,E2 -263.4433} C_DIS
LIN {X 39.0636,Y -2.778,Z 61,A -9.6797,B 24.8445,C -2.8773,E1 25.1596,E2 -267.1782} C_DIS
LIN {X 39.1547,Y 0.7578,Z 61,A -4.8913,B 24.8434,C -2.887,E1 25.1596,E2 -271.9612} C_DIS
LIN {X 39.0459,Y 3.015,Z 61,A -1.6907,B 24.8425,C -2.8956,E1 25.1591,E2 -275.163} C_DIS
LIN {X 38.8804,Y 4.6897,Z 61,A 0.5348,B 24.8421,C -2.8993,E1 25.1584,E2 -277.3841} C_DIS
LIN {X 38.6849,Y 6.0953,Z 61,A 2.5911,B 24.8414,C -2.9053,E1 25.1576,E2 -279.4426} C_DIS
LIN {X 38.2822,Y 8.2549,Z 61,A 6.1686,B 24.8397,C -2.921,E1 25.1556,E2 -283.0365} C_DIS
LIN {X 37.4122,Y 11.5755,Z 61,A 11.5791,B 24.8373,C -2.9423,E1 25.1515,E2 -288.4662} C_DIS
LIN {X 36.6504,Y 13.7991,Z 61,A 14.4294,B 24.8373,C -2.9425,E1 25.1488,E2 -291.3011} C_DIS
LIN {X 35.7872,Y 15.9052,Z 61,A 17.7207,B 24.8363,C -2.9512,E1 25.1452,E2 -294.595} C_DIS
LIN {X 34.648,Y 18.2531,Z 61,A 21.6216,B 24.835,C -2.9629,E1 25.1403,E2 -298.5027} C_DIS
LIN {X 33.547,Y 20.2061,Z 61,A 24.841,B 24.8342,C -2.9704,E1 25.1357,E2 -301.7234} C_DIS
LIN {X 32.3747,Y 22.0345,Z 61,A 28.172,B 24.833,C -2.9808,E1 25.1306,E2 -305.0624} C_DIS
LIN {X 31.276,Y 23.5685,Z 61,A 31.1209,B 24.8319,C -2.9904,E1 25.1256,E2 -308.0199} C_DIS
LIN {X 29.3398,Y 25.9402,Z 61,A 35.0279,B 24.8319,C -2.9915,E1 25.1186,E2 -311.9117} C_DIS
LIN {X 28.1833,Y 27.1911,Z 61,A 38.0113,B 24.8303,C -3.0044,E1 25.1128,E2 -314.9129} C_DIS
LIN {X 26.2053,Y 29.1021,Z 61,A 41.8738,B 24.8297,C -3.0099,E1 25.105,E2 -318.7727} C_DIS
LIN {X 24.1917,Y 30.7967,Z 61,A 45.6485,B 24.8291,C -3.0158,E1 25.0968,E2 -322.5469} C_DIS
LIN {X 21.9599,Y 32.4257,Z 61,A 49.3153,B 24.8289,C -3.0168,E1 25.0884,E2 -326.2034} C_DIS
LIN {X 20.6722,Y 33.2615,Z 61,A 51.7203,B 24.8283,C -3.0225,E1 25.0828,E2 -328.6144} C_DIS
LIN {X 18.856,Y 34.3233,Z 61,A 54.511,B 24.8283,C -3.0225,E1 25.076,E2 -331.3967} C_DIS
LIN {X 17.7501,Y 34.9085,Z 61,A 56.8138,B 24.8272,C -3.0317,E1 25.0702,E2 -333.715} C_DIS
LIN {X 15.4332,Y 35.9935,Z 61,A 60.447,B 24.8269,C -3.0343,E1 25.061,E2 -337.3452} C_DIS
LIN {X 13.2106,Y 36.8672,Z 61,A 64.3159,B 24.826,C -3.0428,E1 25.0508,E2 -341.2261} C_DIS
LIN {X 10.4952,Y 37.7298,Z 61,A 67.922,B 24.8265,C -3.0378,E1 25.0412,E2 -344.8142} C_DIS
LIN {X 8.5401,Y 38.22,Z 61,A 70.9397,B 24.8262,C -3.0404,E1 25.033,E2 -347.8336} C_DIS
LIN {X 6.3398,Y 38.6456,Z 61,A 74.2722,B 24.826,C -3.0423,E1 25.0239,E2 -351.167} C_DIS
LIN {X 2.4637,Y 39.0848,Z 61,A 80.3124,B 24.8254,C -3.0473,E1 25.0071,E2 -357.2156} C_DIS
LIN {X -0.3841,Y 39.1603,Z 61,A 84.0884,B 24.8261,C -3.0415,E1 24.9966,E2 -360.9773} C_DIS
LIN {X -2.5801,Y 39.0767,Z 61,A 86.9614,B 24.8267,C -3.036,E1 24.9886,E2 -363.8379} C_DIS
LIN {X -4.2003,Y 38.9363,Z 61,A 89.8135,B 24.8262,C -3.0408,E1 24.9806,E2 -366.7031} C_DIS
LIN {X -6.5413,Y 38.6119,Z 61,A 93.2096,B 24.8265,C -3.0377,E1 24.9713,E2 -370.0948} C_DIS
LIN {X -9.3284,Y 38.0348,Z 61,A 97.5867,B 24.8267,C -3.0367,E1 24.9593,E2 -374.4751} C_DIS
LIN {X -11.6931,Y 37.3757,Z 61,A 101.4834,B 24.8267,C -3.0366,E1 24.9489,E2 -378.378} C_DIS
LIN {X -15.223,Y 36.0822,Z 61,A 106.4126,B 24.8283,C -3.0225,E1 24.9361,E2 -383.2842} C_DIS
LIN {X -17.5637,Y 35.0028,Z 61,A 110.5761,B 24.8284,C -3.0213,E1 24.9256,E2 -387.4556} C_DIS
LIN {X -19.476,Y 33.9757,Z 61,A 113.1658,B 24.8298,C -3.0092,E1 24.9194,E2 -390.0238} C_DIS
LIN {X -21.1217,Y 32.9778,Z 61,A 116.4018,B 24.8298,C -3.0089,E1 24.9117,E2 -393.2691} C_DIS
LIN {X -23.1867,Y 31.5601,Z 61,A 119.9766,B 24.8308,C -3.0007,E1 24.9035,E2 -396.8367} C_DIS
LIN {X -25.8064,Y 29.4567,Z 61,A 124.5511,B 24.8324,C -2.9864,E1 24.8937,E2 -401.3944} C_DIS
LIN {X -26.7425,Y 28.6097,Z 61,A 126.5675,B 24.8326,C -2.9841,E1 24.8896,E2 -403.4133} C_DIS
LIN {X -27.899,Y 27.4829,Z 61,A 128.9604,B 24.8332,C -2.9789,E1 24.8848,E2 -405.8039} C_DIS
LIN {X -29.0688,Y 26.2426,Z 61,A 131.4584,B 24.8339,C -2.9728,E1 24.8801,E2 -408.2986} C_DIS
LIN {X -30.6226,Y 24.412,Z 61,A 135.0209,B 24.8348,C -2.9645,E1 24.8738,E2 -411.8574} C_DIS
LIN {X -31.9813,Y 22.6011,Z 61,A 138.3844,B 24.8358,C -2.9563,E1 24.8682,E2 -415.2176} C_DIS
LIN {X -33.2218,Y 20.7359,Z 61,A 142.1,B 24.8362,C -2.9519,E1 24.8626,E2 -418.9416} C_DIS
LIN {X -34.4347,Y 18.6525,Z 61,A 145.3532,B 24.8377,C -2.9391,E1 24.8582,E2 -422.1811} C_DIS
LIN {X -35.3596,Y 16.8337,Z 61,A 148.2075,B 24.8388,C -2.9291,E1 24.8546,E2 -425.027} C_DIS
LIN {X -36.0864,Y 15.2129,Z 61,A 150.5887,B 24.8399,C -2.9192,E1 24.852,E2 -427.3976} C_DIS
LIN {X -36.636,Y 13.8372,Z 61,A 153.428,B 24.8399,C -2.9196,E1 24.8491,E2 -430.2538} C_DIS
LIN {X -37.5113,Y 11.2506,Z 61,A 157.1114,B 24.8415,C -2.9043,E1 24.846,E2 -433.9216} C_DIS
LIN {X -38.1199,Y 8.9756,Z 61,A 160.8247,B 24.8424,C -2.8964,E1 24.8435,E2 -437.6377} C_DIS
LIN {X -38.5865,Y 6.6932,Z 61,A 164.0956,B 24.8437,C -2.8844,E1 24.8418,E2 -440.8992} C_DIS
LIN {X -38.8889,Y 4.6172,Z 61,A 167.2721,B 24.8446,C -2.8759,E1 24.8406,E2 -444.0744} C_DIS
Enddeposition()
END
